C05454=1069.423,168.035,-78.116,173.237,27.810,155.027
C05455=1069.428,168.284,-78.138,173.240,27.813,155.027
C05456=1069.434,168.532,-78.160,173.242,27.815,155.028
C05457=1069.440,168.782,-78.182,173.243,27.818,155.028
C05458=1069.445,169.031,-78.205,173.246,27.821,155.028
C05459=1069.452,169.280,-78.227,173.247,27.824,155.029
C05460=1069.457,169.528,-78.250,173.250,27.827,155.029
C05461=1069.462,169.778,-78.272,173.251,27.830,155.030
C05462=1069.468,170.027,-78.294,173.253,27.832,155.030
C05463=1069.473,170.275,-78.316,173.255,27.835,155.030
C05464=1069.479,170.525,-78.338,173.257,27.838,155.031
C05465=1069.485,170.773,-78.361,173.259,27.841,155.031
C05466=1069.491,171.023,-78.383,173.261,27.844,155.032
C05467=1069.496,171.271,-78.405,173.263,27.847,155.032
C05468=1069.502,171.520,-78.427,173.265,27.850,155.032
C05469=1069.508,171.769,-78.450,173.266,27.852,155.033
C05470=1069.513,172.019,-78.472,173.269,27.855,155.033
C05471=1069.519,172.267,-78.495,173.270,27.858,155.034
C05472=1069.525,172.515,-78.517,173.273,27.861,155.034
C05473=1069.530,172.765,-78.539,173.274,27.864,155.034
C05474=1069.536,173.014,-78.562,173.277,27.867,155.035
C05475=1069.542,173.263,-78.584,173.278,27.870,155.035
C05476=1069.548,173.512,-78.607,173.280,27.872,155.036
C05477=1069.553,173.760,-78.630,173.282,27.875,155.036
C05478=1069.558,174.010,-78.652,173.284,27.878,155.036
C05479=1069.565,174.258,-78.674,173.286,27.881,155.037
C05480=1069.570,174.508,-78.696,173.288,27.884,155.037
C05481=1069.576,174.790,-78.722,173.290,27.887,155.037
C05482=1069.583,175.072,-78.747,173.293,27.890,155.038
C05483=1069.590,175.355,-78.774,173.295,27.893,155.038
C05484=1069.597,175.637,-78.799,173.297,27.897,155.039
C05485=1069.602,175.886,-78.821,173.299,27.900,155.039
C05486=1069.608,176.135,-78.844,173.301,27.902,155.040
C05487=1069.614,176.383,-78.866,173.303,27.905,155.040
C05488=1069.619,176.633,-78.888,173.305,27.908,155.040
C05489=1069.625,176.881,-78.911,173.307,27.911,155.041
C05490=1069.631,177.130,-78.934,173.309,27.913,155.041
C05491=1069.637,177.379,-78.957,173.311,27.916,155.042
C05492=1069.642,177.628,-78.979,173.313,27.919,155.042
C05493=1069.648,177.877,-79.002,173.315,27.922,155.042
C05494=1069.654,178.126,-79.025,173.317,27.925,155.043
C05495=1069.660,178.375,-79.048,173.319,27.928,155.043
C05496=1069.666,178.624,-79.070,173.321,27.931,155.044
C05497=1069.672,178.873,-79.092,173.323,27.933,155.044
C05498=1069.677,179.122,-79.115,173.325,27.936,155.044
C05499=1069.682,179.370,-79.138,173.327,27.939,155.045
C05500=1069.688,179.619,-79.161,173.329,27.942,155.045
C05501=1069.695,179.868,-79.183,173.331,27.945,155.046
C05502=1069.700,180.117,-79.206,173.333,27.948,155.046
C05503=1069.706,180.366,-79.229,173.335,27.950,155.046
C05504=1069.711,180.615,-79.251,173.337,27.953,155.047
C05505=1069.717,180.864,-79.274,173.339,27.956,155.047
C05506=1069.724,181.113,-79.296,173.341,27.959,155.048
C05507=1069.729,181.361,-79.319,173.343,27.961,155.048
C05508=1069.735,181.610,-79.342,173.345,27.964,155.048
C05509=1069.741,181.859,-79.365,173.348,27.967,155.049
C05510=1069.747,182.108,-79.388,173.349,27.970,155.049
C05511=1069.753,182.357,-79.411,173.352,27.973,155.049
C05512=1069.759,182.606,-79.434,173.353,27.976,155.050
C05513=1069.765,182.855,-79.456,173.356,27.979,155.050
C05514=1069.770,183.103,-79.479,173.357,27.982,155.051
C05515=1069.777,183.353,-79.503,173.360,27.985,155.051
C05516=1069.782,183.602,-79.526,173.362,27.987,155.051
C05517=1069.788,183.851,-79.549,173.364,27.990,155.052
C05518=1069.795,184.099,-79.571,173.366,27.993,155.052
C05519=1069.800,184.348,-79.594,173.368,27.995,155.052
C05520=1069.806,184.597,-79.617,173.370,27.998,155.053
C05521=1069.812,184.846,-79.640,173.372,28.001,155.053
C05522=1069.817,185.095,-79.663,173.374,28.004,155.054
C05523=1069.822,185.344,-79.686,173.376,28.007,155.054
C05524=1069.828,185.593,-79.709,173.378,28.010,155.055
C05525=1069.834,185.841,-79.733,173.380,28.013,155.055
C05526=1069.839,186.091,-79.756,173.382,28.016,155.055
C05527=1069.845,186.339,-79.779,173.384,28.019,155.056
C05528=1069.851,186.588,-79.802,173.387,28.022,155.056
C05529=1069.856,186.837,-79.825,173.388,28.025,155.057
C05530=1069.861,187.087,-79.849,173.391,28.028,155.057
C05531=1069.867,187.335,-79.872,173.392,28.031,155.057
C05532=1069.873,187.584,-79.895,173.395,28.034,155.058
C05533=1069.878,187.833,-79.919,173.396,28.037,155.058
C05534=1069.884,188.082,-79.942,173.399,28.040,155.059
C05535=1069.890,188.331,-79.965,173.400,28.043,155.059
C05536=1069.896,188.579,-79.989,173.403,28.046,155.060
C05537=1069.901,188.828,-80.012,173.404,28.049,155.060
C05538=1069.906,189.077,-80.035,173.407,28.052,155.060
C05539=1069.912,189.325,-80.059,173.409,28.055,155.061
C05540=1069.917,189.575,-80.082,173.411,28.058,155.061
C05541=1069.923,189.823,-80.105,173.413,28.061,155.062
C05542=1069.929,190.072,-80.128,173.415,28.063,155.062
C05543=1069.934,190.321,-80.152,173.417,28.067,155.063
C05544=1069.940,190.570,-80.175,173.419,28.070,155.063
C05545=1069.946,190.852,-80.202,173.421,28.073,155.063
C05546=1069.952,191.133,-80.228,173.424,28.076,155.064
C05547=1069.959,191.416,-80.255,173.426,28.080,155.064
C05548=1069.965,191.698,-80.282,173.429,28.083,155.065
C05549=1069.971,191.946,-80.305,173.431,28.086,155.065
C05550=1069.977,192.195,-80.328,173.433,28.089,155.066
C05551=1069.982,192.444,-80.352,173.435,28.092,155.066
C05552=1069.988,192.693,-80.376,173.438,28.095,155.066
C05553=1069.994,192.942,-80.399,173.439,28.098,155.067
C05554=1069.999,193.191,-80.423,173.442,28.101,155.067
C05555=1070.005,193.440,-80.446,173.443,28.104,155.068
C05556=1070.011,193.688,-80.470,173.446,28.107,155.068
C05557=1070.016,193.937,-80.493,173.448,28.110,155.069
C05558=1070.022,194.185,-80.517,173.450,28.113,155.069
C05559=1070.027,194.435,-80.540,173.452,28.116,155.069
C05560=1070.034,194.684,-80.565,173.454,28.119,155.070
C05561=1070.040,194.933,-80.587,173.456,28.122,155.070
C05562=1070.045,195.181,-80.612,173.459,28.125,155.071
C05563=1070.051,195.430,-80.635,173.460,28.128,155.071
C05564=1070.056,195.679,-80.659,173.463,28.131,155.072
C05565=1070.062,195.928,-80.682,173.464,28.134,155.072
C05566=1070.068,196.176,-80.706,173.467,28.137,155.072
C05567=1070.074,196.425,-80.730,173.469,28.140,155.073
C05568=1070.079,196.674,-80.753,173.471,28.142,155.073
C05569=1070.085,196.923,-80.777,173.474,28.145,155.074
C05570=1070.091,197.172,-80.801,173.476,28.149,155.074
C05571=1070.097,197.420,-80.824,173.478,28.152,155.074
C05572=1070.102,197.669,-80.849,173.480,28.155,155.075
C05573=1070.108,197.918,-80.872,173.483,28.158,155.075
C05574=1070.114,198.167,-80.896,173.484,28.160,155.076
C05575=1070.120,198.415,-80.920,173.487,28.163,155.076
C05576=1070.125,198.665,-80.943,173.488,28.167,155.077
C05577=1070.131,198.913,-80.967,173.491,28.170,155.077
C05578=1070.137,199.162,-80.992,173.493,28.173,155.077
C05579=1070.143,199.411,-81.015,173.495,28.175,155.078
C05580=1070.149,199.659,-81.038,173.497,28.178,155.078
C05581=1070.154,199.909,-81.063,173.500,28.181,155.079
C05582=1070.161,200.157,-81.087,173.501,28.184,155.079
C05583=1070.166,200.406,-81.111,173.504,28.187,155.079
C05584=1070.172,200.655,-81.134,173.506,28.190,155.080
C05585=1070.177,200.904,-81.158,173.508,28.193,155.080
C05586=1070.183,201.152,-81.182,173.510,28.196,155.081
C05587=1070.189,201.401,-81.207,173.513,28.200,155.081
C05588=1070.195,201.650,-81.230,173.515,28.203,155.082
C05589=1070.200,201.899,-81.254,173.517,28.205,155.082
C05590=1070.207,202.148,-81.278,173.519,28.208,155.082
C05591=1070.212,202.396,-81.302,173.522,28.211,155.083
C05592=1070.218,202.645,-81.326,173.523,28.214,155.083
C05593=1070.224,202.894,-81.350,173.526,28.217,155.084
C05594=1070.230,203.143,-81.375,173.528,28.220,155.084
C05595=1070.235,203.391,-81.399,173.530,28.224,155.085
C05596=1070.241,203.639,-81.423,173.533,28.227,155.085
C05597=1070.247,203.889,-81.446,173.535,28.230,155.085
C05598=1070.252,204.138,-81.471,173.537,28.233,155.086
C05599=1070.257,204.386,-81.495,173.539,28.236,155.086
C05600=1070.264,204.635,-81.519,173.542,28.239,155.087
C05601=1070.269,204.884,-81.543,173.543,28.242,155.087
C05602=1070.274,205.133,-81.568,173.546,28.245,155.088
C05603=1070.280,205.382,-81.592,173.548,28.248,155.088
C05604=1070.286,205.630,-81.616,173.551,28.251,155.088
C05605=1070.292,205.879,-81.640,173.552,28.254,155.089
C05606=1070.297,206.128,-81.665,173.555,28.258,155.089
C05607=1070.303,206.377,-81.689,173.557,28.261,155.090
C05608=1070.309,206.625,-81.714,173.559,28.263,155.090
C05609=1070.338,207.881,-81.837,173.698,28.338,155.093
C05610=1070.343,208.093,-81.858,173.701,28.341,155.094
C05611=1070.348,208.306,-81.880,173.702,28.344,155.094
C05612=1070.353,208.518,-81.901,173.704,28.348,155.095
C05613=1070.359,208.731,-81.923,173.705,28.352,155.096
C05614=1070.363,208.944,-81.944,173.707,28.355,155.096
C05615=1070.368,209.156,-81.966,173.709,28.358,155.097
C05616=1070.373,209.369,-81.987,173.710,28.361,155.097
C05617=1070.379,209.618,-82.012,173.713,28.366,155.098
C05618=1070.385,209.866,-82.037,173.714,28.369,155.099
C05619=1070.391,210.115,-82.062,173.717,28.373,155.099
C05620=1070.397,210.364,-82.087,173.719,28.378,155.100
C05621=1070.402,210.612,-82.113,173.720,28.382,155.101
C05622=1070.409,210.861,-82.138,173.723,28.386,155.101
C05623=1070.414,211.110,-82.163,173.725,28.390,155.102
C05624=1070.420,211.358,-82.188,173.726,28.394,155.103
C05625=1070.426,211.607,-82.213,173.729,28.398,155.103
C05626=1070.432,211.856,-82.239,173.731,28.402,155.104
C05627=1070.437,212.104,-82.264,173.733,28.405,155.104
C05628=1070.444,212.353,-82.289,173.735,28.410,155.105
C05629=1070.449,212.602,-82.314,173.737,28.414,155.106
C05630=1070.456,212.851,-82.339,173.739,28.417,155.106
C05631=1070.461,213.099,-82.365,173.741,28.421,155.107
C05632=1070.467,213.348,-82.390,173.744,28.425,155.108
C05633=1070.473,213.596,-82.416,173.745,28.430,155.108
C05634=1070.478,213.845,-82.442,173.747,28.434,155.109
C05635=1070.484,214.093,-82.467,173.750,28.438,155.110
C05636=1070.490,214.342,-82.492,173.751,28.442,155.110
C05637=1070.496,214.591,-82.518,173.754,28.446,155.111
C05638=1070.502,214.840,-82.543,173.756,28.450,155.112
C05639=1070.508,215.088,-82.568,173.757,28.453,155.112
C05640=1070.513,215.336,-82.594,173.760,28.457,155.113
C05641=1070.519,215.585,-82.619,173.762,28.462,155.114
C05642=1070.525,215.834,-82.645,173.764,28.465,155.114
C05643=1070.531,216.083,-82.671,173.766,28.469,155.115
C05644=1070.537,216.331,-82.696,173.768,28.474,155.116
C05645=1070.543,216.580,-82.722,173.770,28.478,155.116
C05646=1070.548,216.828,-82.747,173.772,28.482,155.117
C05647=1070.554,217.077,-82.772,173.775,28.486,155.118
C05648=1070.560,217.326,-82.798,173.776,28.490,155.118
C05649=1070.566,217.575,-82.824,173.778,28.494,155.119
C05650=1070.572,217.823,-82.850,173.781,28.498,155.119
C05651=1070.578,218.072,-82.875,173.783,28.502,155.120
C05652=1070.584,218.320,-82.901,173.785,28.505,155.121
C05653=1070.590,218.569,-82.927,173.787,28.509,155.121
C05654=1070.595,218.817,-82.952,173.789,28.513,155.122
C05655=1070.601,219.066,-82.978,173.791,28.517,155.123
C05656=1070.607,219.314,-83.004,173.793,28.521,155.123
C05657=1070.613,219.563,-83.029,173.796,28.525,155.124
C05658=1070.619,219.812,-83.055,173.798,28.529,155.125
C05659=1070.625,220.061,-83.080,173.799,28.533,155.125
C05660=1070.631,220.310,-83.106,173.802,28.537,155.126
C05661=1070.637,220.558,-83.132,173.804,28.541,155.127
C05662=1070.643,220.807,-83.158,173.806,28.545,155.127
C05663=1070.649,221.055,-83.184,173.808,28.549,155.128
C05664=1070.655,221.304,-83.209,173.811,28.553,155.129
C05665=1070.660,221.519,-83.232,173.812,28.556,155.129
C05666=1070.665,221.733,-83.254,173.815,28.560,155.130
C05667=1070.670,221.948,-83.277,173.816,28.563,155.130
C05668=1070.675,222.163,-83.298,173.817,28.567,155.131
C05669=1070.680,222.379,-83.322,173.820,28.570,155.131
C05670=1070.685,222.593,-83.344,173.821,28.573,155.132
C05671=1070.690,222.808,-83.367,173.823,28.577,155.132
C05672=1070.695,223.022,-83.389,173.825,28.580,155.133
C05673=1070.701,223.271,-83.415,173.827,28.584,155.134
C05674=1070.707,223.520,-83.440,173.829,28.588,155.134
C05675=1070.713,223.768,-83.467,173.832,28.592,155.135
C05676=1070.718,224.017,-83.493,173.834,28.596,155.136
C05677=1070.725,224.265,-83.519,173.836,28.600,155.136
C05678=1070.730,224.514,-83.545,173.838,28.604,155.137
C05679=1070.736,224.763,-83.571,173.840,28.608,155.138
C05680=1070.741,225.012,-83.597,173.843,28.612,155.138
C05681=1070.748,225.260,-83.623,173.844,28.616,155.139
C05682=1070.753,225.509,-83.649,173.847,28.620,155.139
C05683=1070.759,225.757,-83.676,173.849,28.624,155.140
C05684=1070.765,226.006,-83.701,173.851,28.628,155.141
C05685=1070.771,226.254,-83.728,173.853,28.632,155.141
C05686=1070.776,226.503,-83.754,173.855,28.636,155.142
C05687=1070.783,226.751,-83.780,173.858,28.640,155.143
C05688=1070.788,227.000,-83.806,173.860,28.644,155.143
C05689=1070.794,227.248,-83.833,173.862,28.648,155.144
C05690=1070.800,227.497,-83.859,173.864,28.652,155.145
C05691=1070.806,227.745,-83.885,173.866,28.656,155.145
C05692=1070.812,227.994,-83.911,173.869,28.659,155.146
C05693=1070.817,228.243,-83.937,173.870,28.663,155.146
C05694=1070.825,228.492,-83.964,173.873,28.667,155.147
C05695=1070.830,228.740,-83.990,173.875,28.671,155.148
C05696=1070.836,228.989,-84.016,173.878,28.675,155.148
C05697=1070.842,229.237,-84.043,173.880,28.679,155.149
C05698=1070.848,229.485,-84.069,173.882,28.683,155.150
C05699=1070.854,229.734,-84.095,173.884,28.687,155.150
C05700=1070.859,229.983,-84.121,173.886,28.691,155.151
C05701=1070.865,230.231,-84.148,173.889,28.695,155.152
C05702=1070.871,230.480,-84.175,173.891,28.699,155.152
C05703=1070.877,230.729,-84.201,173.893,28.702,155.153
C05704=1070.883,230.977,-84.228,173.895,28.706,155.154
C05705=1070.888,231.226,-84.254,173.898,28.710,155.154
C05706=1070.894,231.474,-84.281,173.900,28.714,155.155
C05707=1070.901,231.722,-84.307,173.901,28.718,155.155
C05708=1070.906,231.971,-84.333,173.904,28.722,155.156
C05709=1070.912,232.220,-84.360,173.906,28.726,155.157
C05710=1070.918,232.469,-84.387,173.909,28.730,155.157
C05711=1070.924,232.717,-84.413,173.911,28.734,155.158
C05712=1070.930,232.965,-84.440,173.913,28.738,155.159
C05713=1070.936,233.214,-84.467,173.915,28.742,155.159
C05714=1070.941,233.462,-84.493,173.917,28.746,155.160
C05715=1070.947,233.710,-84.520,173.920,28.750,155.161
C05716=1070.953,233.960,-84.546,173.922,28.754,155.161
C05717=1070.959,234.208,-84.573,173.925,28.758,155.162
C05718=1070.965,234.457,-84.599,173.926,28.762,155.163
C05719=1070.971,234.705,-84.626,173.929,28.766,155.163
C05720=1070.976,234.954,-84.653,173.931,28.770,155.164
C05721=1070.981,235.165,-84.676,173.933,28.773,155.164
C05722=1070.986,235.375,-84.698,173.935,28.776,155.165
C05723=1070.991,235.586,-84.722,173.937,28.779,155.165
C05724=1070.996,235.797,-84.744,173.939,28.783,155.166
C05725=1071.001,236.008,-84.767,173.941,28.787,155.167
C05726=1071.006,236.219,-84.789,173.942,28.790,155.167
C05727=1071.011,236.429,-84.812,173.945,28.793,155.168
C05728=1071.016,236.640,-84.836,173.946,28.796,155.168
C05729=1071.022,236.888,-84.862,173.949,28.800,155.169
C05730=1071.028,237.136,-84.889,173.951,28.804,155.170
C05731=1071.033,237.385,-84.916,173.954,28.808,155.170
C05732=1071.040,237.634,-84.943,173.955,28.812,155.171
C05733=1071.045,237.882,-84.969,173.957,28.816,155.172
C05734=1071.050,238.131,-84.997,173.960,28.820,155.172
C05735=1071.057,238.380,-85.024,173.962,28.824,155.173
C05736=1071.063,238.628,-85.051,173.965,28.828,155.173
C05737=1071.069,238.876,-85.078,173.967,28.832,155.174
C05738=1071.074,239.124,-85.104,173.970,28.835,155.175
C05739=1071.081,239.374,-85.131,173.971,28.839,155.175
C05740=1071.087,239.622,-85.158,173.974,28.843,155.176
C05741=1071.092,239.870,-85.186,173.976,28.847,155.177
C05742=1071.098,240.119,-85.213,173.979,28.851,155.177
C05743=1071.104,240.367,-85.240,173.981,28.855,155.178
C05744=1071.110,240.616,-85.266,173.983,28.859,155.178
C05745=1071.117,240.864,-85.294,173.986,28.863,155.179
C05746=1071.122,241.113,-85.321,173.987,28.867,155.180
C05747=1071.127,241.361,-85.348,173.990,28.871,155.180
C05748=1071.134,241.610,-85.376,173.992,28.875,155.181
C05749=1071.140,241.858,-85.402,173.995,28.879,155.182
C05750=1071.146,242.106,-85.429,173.997,28.883,155.182
C05751=1071.152,242.355,-85.457,174.000,28.887,155.183
C05752=1071.157,242.603,-85.484,174.002,28.890,155.184
C05753=1071.163,242.851,-85.511,174.005,28.894,155.184
C05754=1071.169,243.101,-85.539,174.006,28.898,155.185
C05755=1071.175,243.349,-85.565,174.009,28.902,155.185
C05756=1071.180,243.597,-85.593,174.011,28.906,155.186
C05757=1071.187,243.846,-85.620,174.013,28.910,155.187
C05758=1071.193,244.094,-85.648,174.016,28.914,155.188
C05759=1071.198,244.342,-85.675,174.018,28.918,155.188
C05760=1071.204,244.591,-85.703,174.021,28.922,155.189
C05761=1071.209,244.840,-85.730,174.023,28.926,155.189
C05762=1071.216,245.088,-85.758,174.026,28.930,155.190
C05763=1071.221,245.337,-85.785,174.027,28.934,155.191
C05764=1071.227,245.584,-85.812,174.030,28.938,155.191
C05765=1071.234,245.833,-85.839,174.032,28.941,155.192
C05766=1071.239,246.082,-85.867,174.035,28.945,155.193
C05767=1071.246,246.330,-85.895,174.037,28.949,155.193
C05768=1071.251,246.579,-85.922,174.039,28.953,155.194
C05769=1071.257,246.827,-85.950,174.042,28.957,155.194
C05770=1071.262,247.076,-85.977,174.044,28.961,155.195
C05771=1071.268,247.324,-86.005,174.047,28.966,155.196
C05772=1071.274,247.572,-86.033,174.049,28.970,155.197
C05773=1071.279,247.821,-86.060,174.051,28.973,155.197
C05774=1071.285,248.069,-86.088,174.053,28.977,155.198
C05775=1071.291,248.317,-86.116,174.056,28.981,155.199
C05776=1071.297,248.565,-86.144,174.058,28.985,155.199
C05777=1071.306,248.981,-86.189,174.062,28.992,155.200
C05778=1071.316,249.396,-86.237,174.066,28.999,155.201
C05779=1071.326,249.811,-86.283,174.070,29.005,155.202
C05780=1071.335,250.226,-86.329,174.074,29.012,155.204
C05781=1071.341,250.474,-86.357,174.077,29.016,155.204
C05782=1071.347,250.723,-86.385,174.079,29.020,155.205
C05783=1071.353,250.971,-86.412,174.082,29.024,155.206
C05784=1071.359,251.220,-86.441,174.084,29.028,155.206
C05785=1071.365,251.467,-86.468,174.086,29.032,155.207
C05786=1071.371,251.716,-86.496,174.088,29.036,155.207
C05787=1071.376,251.965,-86.524,174.091,29.040,155.208
C05788=1071.382,252.213,-86.551,174.093,29.044,155.209
C05789=1071.388,252.461,-86.579,174.096,29.048,155.209
C05790=1071.394,252.710,-86.608,174.098,29.052,155.210
C05791=1071.399,252.958,-86.636,174.101,29.056,155.211
C05792=1071.406,253.207,-86.663,174.103,29.060,155.211
C05793=1071.412,253.455,-86.692,174.106,29.064,155.212
C05794=1071.417,253.703,-86.720,174.108,29.067,155.213
C05795=1071.423,253.952,-86.748,174.111,29.071,155.213
C05796=1071.429,254.200,-86.775,174.113,29.075,155.214
C05797=1071.435,254.449,-86.804,174.115,29.079,155.215
C05798=1071.440,254.697,-86.832,174.118,29.083,155.215
C05799=1071.446,254.945,-86.860,174.120,29.087,155.216
C05800=1071.453,255.194,-86.888,174.123,29.091,155.217
C05801=1071.458,255.442,-86.916,174.125,29.095,155.217
C05802=1071.464,255.691,-86.944,174.128,29.099,155.218
C05803=1071.470,255.938,-86.973,174.130,29.103,155.218
C05804=1071.476,256.186,-87.000,174.133,29.107,155.219
C05805=1071.482,256.435,-87.029,174.135,29.111,155.220
C05806=1071.488,256.683,-87.057,174.138,29.115,155.220
C05807=1071.494,256.932,-87.085,174.140,29.119,155.221
C05808=1071.500,257.181,-87.113,174.143,29.123,155.222
C05809=1071.506,257.429,-87.141,174.145,29.127,155.222
C05810=1071.512,257.677,-87.170,174.148,29.131,155.223
C05811=1071.518,257.925,-87.198,174.150,29.135,155.224
C05812=1071.523,258.173,-87.226,174.153,29.138,155.224
C05813=1071.529,258.422,-87.254,174.155,29.142,155.225
C05814=1071.535,258.670,-87.283,174.158,29.146,155.225
C05815=1071.541,258.918,-87.311,174.160,29.150,155.226
C05816=1071.547,259.167,-87.339,174.163,29.154,155.227
C05817=1071.553,259.416,-87.367,174.165,29.158,155.227
C05818=1071.560,259.664,-87.396,174.168,29.162,155.228
C05819=1071.565,259.912,-87.424,174.170,29.166,155.229
C05820=1071.571,260.161,-87.453,174.173,29.170,155.229
C05821=1071.578,260.408,-87.481,174.175,29.173,155.230
C05822=1071.584,260.657,-87.510,174.178,29.177,155.231
C05823=1071.589,260.905,-87.537,174.180,29.181,155.231
C05824=1071.595,261.153,-87.567,174.183,29.185,155.232
C05825=1071.601,261.402,-87.595,174.185,29.189,155.233
C05826=1071.608,261.650,-87.624,174.187,29.193,155.233
C05827=1071.614,261.899,-87.652,174.190,29.197,155.234
C05828=1071.620,262.147,-87.680,174.193,29.200,155.234
C05829=1071.630,262.559,-87.727,174.197,29.207,155.235
C05830=1071.640,262.971,-87.775,174.201,29.214,155.237
C05831=1071.651,263.385,-87.822,174.205,29.220,155.238
C05832=1071.661,263.797,-87.870,174.209,29.227,155.239
C05833=1071.665,264.045,-87.899,174.212,29.231,155.239
C05834=1071.671,264.294,-87.927,174.214,29.235,155.240
C05835=1071.678,264.542,-87.956,174.217,29.239,155.241
C05836=1071.684,264.791,-87.985,174.219,29.242,155.241
C05837=1071.690,265.039,-88.014,174.223,29.247,155.242
C05838=1071.695,265.286,-88.043,174.225,29.251,155.243
C05839=1071.701,265.535,-88.071,174.228,29.254,155.243
C05840=1071.707,265.783,-88.100,174.230,29.258,155.244
C05841=1071.713,266.031,-88.129,174.233,29.262,155.245
C05842=1071.719,266.280,-88.158,174.235,29.266,155.245
C05843=1071.725,266.528,-88.186,174.238,29.270,155.246
C05844=1071.730,266.776,-88.216,174.240,29.274,155.246
C05845=1071.736,267.025,-88.244,174.243,29.278,155.247
C05846=1071.743,267.273,-88.273,174.245,29.282,155.248
C05847=1071.749,267.521,-88.302,174.248,29.286,155.249
C05848=1071.754,267.769,-88.332,174.250,29.290,155.249
C05849=1071.760,268.018,-88.360,174.253,29.294,155.250
C05850=1071.766,268.266,-88.389,174.255,29.298,155.251
C05851=1071.772,268.514,-88.418,174.258,29.302,155.251
C05852=1071.778,268.762,-88.447,174.261,29.306,155.252
C05853=1071.784,269.010,-88.477,174.264,29.310,155.252
C05854=1071.790,269.258,-88.506,174.266,29.314,155.253
C05855=1071.796,269.507,-88.534,174.269,29.318,155.254
C05856=1071.802,269.756,-88.564,174.271,29.322,155.254
C05857=1071.808,270.004,-88.593,174.274,29.326,155.255
C05858=1071.814,270.252,-88.622,174.276,29.330,155.256
C05859=1071.819,270.500,-88.651,174.279,29.334,155.256
C05860=1071.825,270.748,-88.680,174.281,29.338,155.257
C05861=1071.831,270.996,-88.709,174.284,29.342,155.258
C05862=1071.837,271.244,-88.739,174.286,29.346,155.258
C05863=1071.843,271.493,-88.768,174.290,29.350,155.259
C05864=1071.849,271.741,-88.798,174.292,29.354,155.260
C05865=1071.855,271.989,-88.827,174.295,29.358,155.260
C05866=1071.861,272.237,-88.856,174.297,29.362,155.261
C05867=1071.867,272.486,-88.885,174.300,29.366,155.262
C05868=1071.873,272.734,-88.914,174.302,29.370,155.262
C05869=1071.879,272.982,-88.944,174.305,29.374,155.263
C05870=1071.885,273.230,-88.973,174.307,29.378,155.264
C05871=1071.891,273.479,-89.002,174.310,29.382,155.264
C05872=1071.897,273.727,-89.032,174.313,29.386,155.265
C05873=1071.903,273.974,-89.061,174.316,29.390,155.266
C05874=1071.909,274.223,-89.091,174.318,29.394,155.266
C05875=1071.915,274.471,-89.120,174.321,29.398,155.267
C05876=1071.920,274.719,-89.150,174.323,29.402,155.268
C05877=1071.926,274.968,-89.179,174.326,29.406,155.268
C05878=1071.932,275.216,-89.208,174.328,29.410,155.269
C05879=1071.938,275.464,-89.239,174.332,29.414,155.270
C05880=1071.944,275.712,-89.268,174.334,29.418,155.270
C05881=1071.953,276.128,-89.317,174.338,29.425,155.271
C05882=1071.964,276.544,-89.367,174.342,29.432,155.273
C05883=1071.973,276.959,-89.417,174.347,29.438,155.274
C05884=1071.983,277.375,-89.466,174.352,29.445,155.275
C05885=1071.989,277.623,-89.496,174.354,29.449,155.276
C05886=1071.995,277.871,-89.525,174.357,29.453,155.276
C05887=1072.001,278.120,-89.555,174.359,29.457,155.277
C05888=1072.007,278.368,-89.586,174.362,29.461,155.278
C05889=1072.014,278.616,-89.615,174.365,29.465,155.278
C05890=1072.019,278.864,-89.645,174.368,29.470,155.279
C05891=1072.025,279.113,-89.675,174.370,29.474,155.280
C05892=1072.031,279.361,-89.704,174.373,29.477,155.280
C05893=1072.037,279.609,-89.734,174.375,29.481,155.281
C05894=1072.043,279.857,-89.764,174.378,29.485,155.282
C05895=1072.049,280.105,-89.793,174.381,29.490,155.282
C05896=1072.055,280.353,-89.823,174.384,29.494,155.283
C05897=1072.061,280.602,-89.854,174.386,29.498,155.284
C05898=1072.067,280.850,-89.883,174.389,29.502,155.284
C05899=1072.073,281.098,-89.913,174.391,29.506,155.285
C05900=1072.079,281.345,-89.943,174.394,29.510,155.286
C05901=1072.084,281.594,-89.973,174.397,29.514,155.286
C05902=1072.090,281.842,-90.003,174.400,29.518,155.287
C05903=1072.096,282.090,-90.033,174.402,29.522,155.288
C05904=1072.102,282.338,-90.063,174.405,29.526,155.288
C05905=1072.109,282.586,-90.094,174.408,29.530,155.289
C05906=1072.114,282.835,-90.123,174.411,29.535,155.290
C05907=1072.120,283.082,-90.154,174.414,29.539,155.290
C05908=1072.126,283.330,-90.184,174.416,29.543,155.291
C05909=1072.131,283.579,-90.214,174.419,29.546,155.292
C05910=1072.137,283.826,-90.244,174.421,29.551,155.293
C05911=1072.144,284.075,-90.275,174.425,29.555,155.293
C05912=1072.149,284.323,-90.305,174.427,29.559,155.294
C05913=1072.155,284.571,-90.335,174.430,29.563,155.295
C05914=1072.162,284.819,-90.364,174.432,29.567,155.295
C05915=1072.167,285.067,-90.395,174.436,29.571,155.296
C05916=1072.174,285.315,-90.425,174.438,29.576,155.297
C05917=1072.180,285.563,-90.456,174.441,29.580,155.297
C05918=1072.185,285.811,-90.485,174.443,29.583,155.298
C05919=1072.191,286.059,-90.516,174.446,29.587,155.299
C05920=1072.197,286.308,-90.546,174.449,29.592,155.299
C05921=1072.203,286.555,-90.577,174.452,29.596,155.300
C05922=1072.209,286.803,-90.607,174.454,29.600,155.301
C05923=1072.215,287.051,-90.638,174.457,29.604,155.302
C05924=1072.221,287.300,-90.668,174.460,29.608,155.302
C05925=1072.227,287.547,-90.699,174.463,29.612,155.303
C05926=1072.233,287.795,-90.729,174.465,29.617,155.304
C05927=1072.239,288.044,-90.760,174.468,29.620,155.304
C05928=1072.246,288.291,-90.789,174.471,29.625,155.305
C05929=1072.252,288.539,-90.820,174.474,29.628,155.306
C05930=1072.257,288.787,-90.850,174.476,29.633,155.306
C05931=1072.264,289.035,-90.881,174.479,29.637,155.307
C05932=1072.269,289.284,-90.912,174.483,29.641,155.308
C05933=1072.274,289.497,-90.937,174.484,29.644,155.308
C05934=1072.279,289.710,-90.964,174.487,29.648,155.309
C05935=1072.285,289.923,-90.990,174.489,29.652,155.310
C05936=1072.289,290.136,-91.016,174.492,29.655,155.310
C05937=1072.295,290.349,-91.043,174.494,29.659,155.311
C05938=1072.300,290.562,-91.069,174.496,29.662,155.311
C05939=1072.305,290.774,-91.095,174.499,29.666,155.312
C05940=1072.310,290.989,-91.122,174.501,29.669,155.312
C05941=1072.316,291.236,-91.153,174.504,29.674,155.313
C05942=1072.322,291.484,-91.183,174.507,29.678,155.314
C05943=1072.328,291.732,-91.214,174.510,29.682,155.315
C05944=1072.334,291.980,-91.244,174.512,29.686,155.315
C05945=1072.340,292.228,-91.275,174.515,29.690,155.316
C05946=1072.346,292.476,-91.307,174.518,29.694,155.317
C05947=1072.352,292.724,-91.337,174.521,29.698,155.317
C05948=1072.358,292.972,-91.368,174.523,29.703,155.318
C05949=1072.364,293.219,-91.399,174.527,29.707,155.319
C05950=1072.369,293.468,-91.430,174.529,29.711,155.320
C05951=1072.376,293.716,-91.460,174.532,29.715,155.320
C05952=1072.381,293.964,-91.491,174.535,29.720,155.321
C05953=1072.388,294.212,-91.522,174.538,29.724,155.322
C05954=1072.394,294.460,-91.553,174.541,29.728,155.322
C05955=1072.400,294.708,-91.585,174.543,29.732,155.323
C05956=1072.406,294.956,-91.615,174.547,29.736,155.324
C05957=1072.412,295.204,-91.645,174.549,29.740,155.325
C05958=1072.418,295.452,-91.677,174.552,29.745,155.325
C05959=1072.423,295.700,-91.708,174.555,29.749,155.326
C05960=1072.430,295.947,-91.739,174.558,29.753,155.327
C05961=1072.435,296.196,-91.770,174.560,29.757,155.327
C05962=1072.442,296.444,-91.801,174.564,29.762,155.328
C05963=1072.448,296.691,-91.832,174.566,29.766,155.329
C05964=1072.454,296.940,-91.864,174.569,29.770,155.330
C05965=1072.460,297.187,-91.894,174.572,29.774,155.330
C05966=1072.466,297.435,-91.926,174.575,29.778,155.331
C05967=1072.471,297.683,-91.957,174.577,29.782,155.332
C05968=1072.477,297.932,-91.989,174.581,29.787,155.332
C05969=1072.484,298.179,-92.020,174.583,29.791,155.333
C05970=1072.489,298.427,-92.051,174.586,29.796,155.334
C05971=1072.495,298.675,-92.082,174.590,29.800,155.335
C05972=1072.501,298.922,-92.114,174.592,29.804,155.335
C05973=1072.506,299.171,-92.145,174.595,29.808,155.336
C05974=1072.513,299.418,-92.176,174.598,29.813,155.337
C05975=1072.519,299.667,-92.208,174.601,29.817,155.338
C05976=1072.524,299.915,-92.239,174.603,29.821,155.338
C05977=1072.530,300.163,-92.271,174.607,29.826,155.339
C05978=1072.536,300.410,-92.302,174.609,29.830,155.340
C05979=1072.542,300.658,-92.334,174.612,29.834,155.341
C05980=1072.548,300.906,-92.365,174.615,29.839,155.341
C05981=1072.553,301.154,-92.397,174.618,29.843,155.342
C05982=1072.560,301.402,-92.428,174.621,29.847,155.343
C05983=1072.566,301.650,-92.460,174.624,29.852,155.344
C05984=1072.571,301.897,-92.491,174.626,29.856,155.344
C05985=1072.578,302.145,-92.523,174.630,29.861,155.345
C05986=1072.583,302.393,-92.554,174.632,29.864,155.346
C05987=1072.589,302.641,-92.586,174.635,29.869,155.347
C05988=1072.595,302.890,-92.618,174.638,29.873,155.347
C05989=1072.600,303.109,-92.646,174.641,29.877,155.348
C05990=1072.606,303.330,-92.673,174.644,29.881,155.349
C05991=1072.611,303.550,-92.702,174.646,29.885,155.349
C05992=1072.616,303.771,-92.730,174.649,29.889,155.350
C05993=1072.621,303.991,-92.759,174.651,29.893,155.351
C05994=1072.627,304.211,-92.787,174.654,29.896,155.351
C05995=1072.632,304.431,-92.815,174.657,29.900,155.352
C05996=1072.637,304.651,-92.843,174.659,29.904,155.353
C05997=1072.643,304.900,-92.875,174.662,29.908,155.353
C05998=1072.650,305.148,-92.907,174.665,29.913,155.354
C05999=1072.655,305.395,-92.938,174.668,29.917,155.355
C06000=1072.661,305.643,-92.970,174.671,29.921,155.356
C06001=1072.667,305.892,-93.002,174.674,29.926,155.356
C06002=1072.673,306.139,-93.034,174.677,29.930,155.357
C06003=1072.679,306.387,-93.066,174.680,29.935,155.358
C06004=1072.685,306.635,-93.098,174.682,29.939,155.359
C06005=1072.691,306.882,-93.130,174.686,29.943,155.359
C06006=1072.698,307.130,-93.161,174.689,29.948,155.360
C06007=1072.704,307.378,-93.193,174.692,29.952,155.361
C06008=1072.710,307.626,-93.225,174.695,29.957,155.362
C06009=1072.715,307.874,-93.257,174.698,29.961,155.362
C06010=1072.722,308.121,-93.289,174.701,29.965,155.363
C06011=1072.728,308.369,-93.321,174.704,29.969,155.364
C06012=1072.734,308.618,-93.353,174.707,29.974,155.365
C06013=1072.740,308.866,-93.385,174.709,29.978,155.366
C06014=1072.746,309.113,-93.418,174.713,29.983,155.366
C06015=1072.753,309.361,-93.449,174.715,29.987,155.367
C06016=1072.759,309.609,-93.481,174.719,29.991,155.368
C06017=1072.765,309.856,-93.514,174.721,29.996,155.369
C06018=1072.771,310.105,-93.546,174.725,30.000,155.369
C06019=1072.776,310.352,-93.578,174.728,30.004,155.370
C06020=1072.783,310.599,-93.610,174.731,30.009,155.371
C06021=1072.789,310.848,-93.642,174.734,30.013,155.371
C06022=1072.796,311.095,-93.675,174.737,30.017,155.372
C06023=1072.802,311.343,-93.707,174.740,30.022,155.373
C06024=1072.808,311.592,-93.739,174.743,30.026,155.374
C06025=1072.814,311.839,-93.771,174.746,30.031,155.375
C06026=1072.820,312.087,-93.803,174.749,30.035,155.375
C06027=1072.827,312.335,-93.836,174.752,30.040,155.376
C06028=1072.832,312.582,-93.867,174.755,30.044,155.377
C06029=1072.838,312.830,-93.900,174.758,30.048,155.378
C06030=1072.844,313.078,-93.932,174.762,30.053,155.378
C06031=1072.851,313.326,-93.965,174.764,30.057,155.379
C06032=1072.857,313.573,-93.997,174.768,30.061,155.380
C06033=1072.863,313.821,-94.029,174.770,30.066,155.381
C06034=1072.869,314.069,-94.062,174.774,30.070,155.381
C06035=1072.875,314.317,-94.094,174.776,30.075,155.382
C06036=1072.882,314.565,-94.127,174.780,30.079,155.383
C06037=1072.888,314.812,-94.160,174.782,30.084,155.384
C06038=1072.894,315.061,-94.192,174.786,30.088,155.385
C06039=1072.899,315.309,-94.225,174.788,30.093,155.386
C06040=1072.906,315.556,-94.258,174.792,30.098,155.386
C06041=1072.912,315.804,-94.291,174.795,30.102,155.387
C06042=1072.917,316.052,-94.323,174.798,30.106,155.388
C06043=1072.923,316.299,-94.356,174.801,30.111,155.389
C06044=1072.929,316.547,-94.388,174.804,30.116,155.390
C06045=1072.934,316.769,-94.418,174.807,30.120,155.390
C06046=1072.940,316.991,-94.448,174.809,30.124,155.391
C06047=1072.945,317.213,-94.476,174.812,30.128,155.392
C06048=1072.950,317.435,-94.506,174.815,30.132,155.392
C06049=1072.955,317.657,-94.536,174.817,30.137,155.393
C06050=1072.961,317.879,-94.565,174.820,30.140,155.394
C06051=1072.966,318.101,-94.594,174.823,30.145,155.395
C06052=1072.972,318.324,-94.624,174.826,30.149,155.395
C06053=1072.978,318.571,-94.657,174.828,30.154,155.396
C06054=1072.984,318.819,-94.691,174.832,30.158,155.397
C06055=1072.990,319.067,-94.723,174.835,30.162,155.398
C06056=1072.996,319.314,-94.756,174.838,30.168,155.399
C06057=1073.002,319.562,-94.789,174.841,30.172,155.400
C06058=1073.008,319.810,-94.822,174.844,30.176,155.400
C06059=1073.014,320.058,-94.855,174.848,30.181,155.401
C06060=1073.020,320.305,-94.888,174.850,30.186,155.402
C06061=1073.026,320.553,-94.921,174.854,30.190,155.403
C06062=1073.032,320.801,-94.954,174.856,30.195,155.404
C06063=1073.038,321.049,-94.987,174.860,30.200,155.404
C06064=1073.044,321.296,-95.020,174.862,30.204,155.405
C06065=1073.050,321.544,-95.053,174.866,30.209,155.406
C06066=1073.056,321.792,-95.086,174.869,30.213,155.407
C06067=1073.062,322.040,-95.119,174.872,30.219,155.408
C06068=1073.069,322.287,-95.153,174.876,30.223,155.409
C06069=1073.075,322.535,-95.186,174.878,30.227,155.409
C06070=1073.081,322.783,-95.219,174.882,30.232,155.410
C06071=1073.087,323.031,-95.252,174.884,30.237,155.411
C06072=1073.093,323.278,-95.285,174.888,30.242,155.412
C06073=1073.099,323.526,-95.319,174.891,30.246,155.413
C06074=1073.105,323.773,-95.352,174.894,30.251,155.414
C06075=1073.111,324.022,-95.386,174.897,30.256,155.414
C06076=1073.117,324.269,-95.418,174.900,30.261,155.415
C06077=1073.123,324.517,-95.452,174.904,30.265,155.416
C06078=1073.130,324.764,-95.485,174.907,30.270,155.417
C06079=1073.135,325.012,-95.519,174.910,30.274,155.418
C06080=1073.142,325.260,-95.552,174.913,30.279,155.419
C06081=1073.148,325.508,-95.586,174.916,30.284,155.419
C06082=1073.155,325.755,-95.619,174.919,30.288,155.420
C06083=1073.160,326.003,-95.652,174.923,30.293,155.421
C06084=1073.167,326.251,-95.686,174.925,30.298,155.422
C06085=1073.173,326.498,-95.720,174.929,30.303,155.423
C06086=1073.178,326.746,-95.753,174.933,30.307,155.424
C06087=1073.186,326.994,-95.787,174.935,30.312,155.425
C06088=1073.191,327.242,-95.820,174.939,30.317,155.425
C06089=1073.198,327.489,-95.854,174.942,30.322,155.426
C06090=1073.204,327.737,-95.887,174.945,30.326,155.427
C06091=1073.210,327.984,-95.921,174.948,30.331,155.428
C06092=1073.216,328.232,-95.954,174.951,30.336,155.429
C06093=1073.223,328.480,-95.988,174.955,30.340,155.430
C06094=1073.229,328.727,-96.022,174.958,30.345,155.431
C06095=1073.235,328.975,-96.055,174.961,30.350,155.431
C06096=1073.242,329.223,-96.089,174.964,30.355,155.432
C06097=1073.247,329.471,-96.122,174.968,30.360,155.433
C06098=1073.255,329.718,-96.156,174.970,30.364,155.434
C06099=1073.260,329.965,-96.190,174.974,30.369,155.435
C06100=1073.266,330.213,-96.224,174.977,30.374,155.436
C06101=1073.272,330.432,-96.253,174.980,30.378,155.436
C06102=1073.278,330.651,-96.284,174.983,30.382,155.437
C06103=1073.284,330.870,-96.314,174.986,30.387,155.438
C06104=1073.289,331.089,-96.343,174.989,30.391,155.439
C06105=1073.295,331.308,-96.373,174.992,30.395,155.439
C06106=1073.300,331.527,-96.403,174.994,30.399,155.440
C06107=1073.306,331.745,-96.433,174.998,30.404,155.441
C06108=1073.311,331.964,-96.464,175.000,30.408,155.442
C06109=1073.317,332.212,-96.497,175.004,30.413,155.443
C06110=1073.323,332.460,-96.531,175.006,30.418,155.444
C06111=1073.329,332.707,-96.565,175.010,30.423,155.445
C06112=1073.336,332.955,-96.600,175.014,30.428,155.445
C06113=1073.341,333.202,-96.634,175.016,30.433,155.446
C06114=1073.347,333.450,-96.668,175.020,30.438,155.447
C06115=1073.354,333.698,-96.702,175.023,30.443,155.448
C06116=1073.360,333.945,-96.736,175.027,30.448,155.449
C06117=1073.366,334.193,-96.771,175.029,30.452,155.450
C06118=1073.372,334.440,-96.805,175.033,30.457,155.451
C06119=1073.378,334.688,-96.839,175.036,30.463,155.452
C06120=1073.384,334.936,-96.873,175.039,30.467,155.453
C06121=1073.391,335.184,-96.908,175.043,30.472,155.454
C06122=1073.397,335.431,-96.942,175.046,30.477,155.454
C06123=1073.403,335.679,-96.976,175.050,30.482,155.455
C06124=1073.409,335.926,-97.010,175.052,30.487,155.456
C06125=1073.416,336.173,-97.045,175.056,30.492,155.457
C06126=1073.422,336.421,-97.079,175.059,30.497,155.458
C06127=1073.428,336.669,-97.114,175.063,30.502,155.459
C06128=1073.434,336.916,-97.148,175.066,30.508,155.460
C06129=1073.440,337.164,-97.182,175.069,30.513,155.461
C06130=1073.447,337.412,-97.217,175.073,30.518,155.462
C06131=1073.453,337.659,-97.251,175.076,30.523,155.463
C06132=1073.459,337.907,-97.286,175.080,30.528,155.464
C06133=1073.465,338.154,-97.320,175.082,30.532,155.465
C06134=1073.472,338.401,-97.355,175.086,30.538,155.466
C06135=1073.477,338.649,-97.390,175.089,30.543,155.467
C06136=1073.484,338.897,-97.424,175.093,30.548,155.467
C06137=1073.490,339.144,-97.459,175.096,30.553,155.468
C06138=1073.496,339.391,-97.493,175.099,30.558,155.469
C06139=1073.502,339.640,-97.528,175.103,30.563,155.470
C06140=1073.508,339.886,-97.563,175.106,30.568,155.471
C06141=1073.515,340.134,-97.598,175.110,30.574,155.472
C06142=1073.521,340.382,-97.633,175.112,30.579,155.473
C06143=1073.526,340.629,-97.667,175.116,30.584,155.474
C06144=1073.533,340.877,-97.702,175.120,30.589,155.475
C06145=1073.540,341.125,-97.737,175.123,30.594,155.476
C06146=1073.546,341.371,-97.772,175.127,30.600,155.477
C06147=1073.552,341.620,-97.807,175.129,30.604,155.478
C06148=1073.558,341.867,-97.842,175.133,30.610,155.479
C06149=1073.564,342.114,-97.876,175.136,30.615,155.480
C06150=1073.571,342.362,-97.911,175.140,30.620,155.481
C06151=1073.577,342.609,-97.947,175.144,30.625,155.482
C06152=1073.583,342.857,-97.981,175.147,30.630,155.483
C06153=1073.590,343.104,-98.016,175.150,30.636,155.484
C06154=1073.596,343.352,-98.052,175.153,30.641,155.485
C06155=1073.602,343.600,-98.086,175.157,30.646,155.486
C06156=1073.608,343.846,-98.121,175.160,30.651,155.487
C06157=1073.614,344.063,-98.152,175.163,30.656,155.488
C06158=1073.619,344.279,-98.182,175.167,30.660,155.488
C06159=1073.625,344.496,-98.214,175.169,30.665,155.489
C06160=1073.630,344.711,-98.244,175.172,30.670,155.490
C06161=1073.635,344.929,-98.274,175.176,30.674,155.491
C06162=1073.641,345.144,-98.305,175.178,30.679,155.492
C06163=1073.647,345.361,-98.336,175.182,30.684,155.493
C06164=1073.651,345.577,-98.367,175.184,30.688,155.494
C06165=1073.658,345.825,-98.402,175.188,30.694,155.495
C06166=1073.664,346.072,-98.438,175.192,30.699,155.496
C06167=1073.671,346.320,-98.473,175.195,30.704,155.497
C06168=1073.676,346.567,-98.508,175.198,30.710,155.498
C06169=1073.683,346.814,-98.543,175.201,30.715,155.499
C06170=1073.689,347.062,-98.579,175.205,30.721,155.500
C06171=1073.696,347.309,-98.614,175.208,30.726,155.501
C06172=1073.702,347.557,-98.650,175.212,30.731,155.502
C06173=1073.709,347.804,-98.685,175.216,30.737,155.503
C06174=1073.714,348.051,-98.720,175.219,30.742,155.504
C06175=1073.721,348.298,-98.755,175.223,30.748,155.505
C06176=1073.727,348.546,-98.791,175.226,30.753,155.506
C06177=1073.733,348.794,-98.827,175.230,30.759,155.507
C06178=1073.740,349.041,-98.862,175.232,30.764,155.508
C06179=1073.746,349.289,-98.898,175.236,30.769,155.509
C06180=1073.752,349.536,-98.934,175.240,30.775,155.510
C06181=1073.758,349.783,-98.969,175.243,30.780,155.511
C06182=1073.764,350.030,-99.005,175.247,30.786,155.512
C06183=1073.770,350.278,-99.040,175.250,30.791,155.513
C06184=1073.777,350.525,-99.076,175.254,30.797,155.514
C06185=1073.783,350.772,-99.112,175.258,30.802,155.515
C06186=1073.790,351.020,-99.147,175.261,30.808,155.516
C06187=1073.796,351.267,-99.183,175.265,30.813,155.517
C06188=1073.803,351.514,-99.219,175.268,30.819,155.518
C06189=1073.809,351.762,-99.254,175.272,30.824,155.519
C06190=1073.815,352.009,-99.290,175.275,30.830,155.520
C06191=1073.822,352.257,-99.327,175.279,30.835,155.521
C06192=1073.828,352.504,-99.362,175.283,30.841,155.522
C06193=1073.835,352.752,-99.398,175.286,30.847,155.524
C06194=1073.841,352.999,-99.434,175.290,30.852,155.525
C06195=1073.847,353.246,-99.470,175.293,30.857,155.526
C06196=1073.853,353.493,-99.506,175.297,30.863,155.527
C06197=1073.859,353.741,-99.542,175.301,30.869,155.528
C06198=1073.866,353.988,-99.578,175.304,30.874,155.529
C06199=1073.872,354.236,-99.614,175.308,30.880,155.530
C06200=1073.879,354.483,-99.650,175.310,30.886,155.531
C06201=1073.885,354.730,-99.686,175.314,30.891,155.532
C06202=1073.891,354.977,-99.722,175.318,30.897,155.533
C06203=1073.897,355.224,-99.759,175.321,30.903,155.534
C06204=1073.903,355.472,-99.794,175.325,30.909,155.535
C06205=1073.910,355.719,-99.831,175.328,30.914,155.536
C06206=1073.916,355.966,-99.867,175.333,30.920,155.538
C06207=1073.922,356.214,-99.903,175.336,30.926,155.539
C06208=1073.928,356.461,-99.939,175.340,30.932,155.540
C06209=1073.935,356.708,-99.976,175.344,30.937,155.541
C06210=1073.941,356.956,-100.012,175.347,30.943,155.542
C06211=1073.948,357.203,-100.048,175.351,30.948,155.543
C06212=1073.954,357.450,-100.085,175.354,30.954,155.544
C06213=1073.960,357.668,-100.116,175.357,30.959,155.545
C06214=1073.965,357.886,-100.149,175.361,30.965,155.546
C06215=1073.971,358.104,-100.181,175.363,30.969,155.547
C06216=1073.977,358.322,-100.212,175.367,30.975,155.548
C06217=1073.983,358.541,-100.245,175.371,30.980,155.549
C06218=1073.988,358.759,-100.277,175.373,30.985,155.550
C06219=1073.994,358.976,-100.309,175.377,30.990,155.551
C06220=1073.999,359.195,-100.342,175.380,30.995,155.552
C06221=1074.006,359.442,-100.378,175.383,31.001,155.553
C06222=1074.012,359.689,-100.414,175.387,31.007,155.554
C06223=1074.018,359.936,-100.451,175.390,31.013,155.556
C06224=1074.025,360.183,-100.487,175.395,31.019,155.557
C06225=1074.032,360.431,-100.524,175.399,31.025,155.558
C06226=1074.038,360.678,-100.561,175.402,31.031,155.559
C06227=1074.044,360.925,-100.597,175.406,31.037,155.560
C06228=1074.050,361.172,-100.634,175.409,31.042,155.561
C06229=1074.057,361.419,-100.672,175.413,31.048,155.563
C06230=1074.064,361.666,-100.708,175.417,31.054,155.564
C06231=1074.070,361.914,-100.744,175.420,31.060,155.565
C06232=1074.076,362.161,-100.781,175.424,31.066,155.566
C06233=1074.083,362.408,-100.818,175.427,31.072,155.567
C06234=1074.089,362.656,-100.855,175.431,31.078,155.568
C06235=1074.095,362.902,-100.892,175.436,31.084,155.569
C06236=1074.102,363.149,-100.928,175.439,31.090,155.571
C06237=1074.109,363.397,-100.965,175.443,31.096,155.572
C06238=1074.115,363.644,-101.003,175.446,31.102,155.573
C06239=1074.121,363.891,-101.039,175.450,31.108,155.574
C06240=1074.128,364.139,-101.076,175.454,31.114,155.575
C06241=1074.135,364.385,-101.113,175.457,31.120,155.577
C06242=1074.140,364.632,-101.150,175.461,31.126,155.578
C06243=1074.147,364.880,-101.187,175.465,31.133,155.579
C06244=1074.154,365.127,-101.224,175.469,31.138,155.580
C06245=1074.160,365.375,-101.262,175.473,31.145,155.581
C06246=1074.167,365.621,-101.299,175.476,31.151,155.583
C06247=1074.172,365.868,-101.336,175.480,31.157,155.584
C06248=1074.179,366.116,-101.373,175.483,31.163,155.585
C06249=1074.186,366.362,-101.411,175.487,31.170,155.586
C06250=1074.192,366.609,-101.448,175.492,31.176,155.587
C06251=1074.199,366.856,-101.485,175.495,31.182,155.589
C06252=1074.205,367.104,-101.522,175.499,31.188,155.590
C06253=1074.211,367.350,-101.559,175.503,31.195,155.591
C06254=1074.218,367.598,-101.598,175.506,31.201,155.592
C06255=1074.224,367.845,-101.634,175.511,31.207,155.594
C06256=1074.231,368.092,-101.672,175.514,31.214,155.595
C06257=1074.237,368.339,-101.709,175.518,31.220,155.596
C06258=1074.244,368.586,-101.747,175.522,31.226,155.597
C06259=1074.250,368.833,-101.784,175.525,31.232,155.599
C06260=1074.256,369.080,-101.822,175.530,31.238,155.600
C06261=1074.263,369.327,-101.859,175.533,31.245,155.601
C06262=1074.269,369.574,-101.897,175.537,31.251,155.602
C06263=1074.276,369.821,-101.934,175.541,31.258,155.604
C06264=1074.282,370.068,-101.971,175.544,31.264,155.605
C06265=1074.288,370.316,-102.010,175.549,31.270,155.606
C06266=1074.295,370.562,-102.047,175.553,31.277,155.608
C06267=1074.302,370.810,-102.085,175.556,31.283,155.609
C06268=1074.309,371.057,-102.122,175.560,31.290,155.610
C06269=1074.315,371.324,-102.164,175.564,31.297,155.612
C06270=1074.323,371.592,-102.204,175.569,31.304,155.613
C06271=1074.329,371.859,-102.245,175.573,31.310,155.614
C06272=1074.337,372.126,-102.286,175.577,31.317,155.616
C06273=1074.344,372.373,-102.324,175.581,31.324,155.617
C06274=1074.350,372.620,-102.361,175.585,31.330,155.618
C06275=1074.357,372.867,-102.400,175.589,31.337,155.620
C06276=1074.363,373.114,-102.437,175.593,31.343,155.621
C06277=1074.370,373.361,-102.475,175.596,31.350,155.622
C06278=1074.376,373.608,-102.513,175.600,31.357,155.624
C06279=1074.383,373.855,-102.551,175.605,31.363,155.625
C06280=1074.389,374.102,-102.590,175.608,31.370,155.626
C06281=1074.396,374.348,-102.627,175.612,31.376,155.628
C06282=1074.402,374.596,-102.665,175.616,31.383,155.629
C06283=1074.409,374.843,-102.704,175.620,31.390,155.630
C06284=1074.415,375.089,-102.741,175.624,31.396,155.632
C06285=1074.422,375.337,-102.780,175.628,31.403,155.633
C06286=1074.428,375.584,-102.818,175.632,31.410,155.634
C06287=1074.434,375.831,-102.856,175.636,31.417,155.636
C06288=1074.441,376.077,-102.895,175.639,31.423,155.637
C06289=1074.448,376.324,-102.932,175.644,31.430,155.638
C06290=1074.455,376.571,-102.971,175.648,31.437,155.640
C06291=1074.461,376.818,-103.009,175.651,31.444,155.641
C06292=1074.468,377.065,-103.048,175.656,31.450,155.642
C06293=1074.474,377.312,-103.086,175.660,31.457,155.644
C06294=1074.481,377.558,-103.124,175.663,31.464,155.645
C06295=1074.487,377.806,-103.163,175.668,31.471,155.647
C06296=1074.494,378.053,-103.201,175.672,31.477,155.648
C06297=1074.501,378.300,-103.240,175.675,31.484,155.649
C06298=1074.507,378.546,-103.278,175.680,31.491,155.651
C06299=1074.513,378.793,-103.317,175.684,31.498,155.652
C06300=1074.520,379.040,-103.356,175.687,31.505,155.654
C06301=1074.527,379.287,-103.393,175.692,31.512,155.655
C06302=1074.534,379.534,-103.432,175.696,31.519,155.656
C06303=1074.540,379.780,-103.471,175.700,31.526,155.658
C06304=1074.547,380.027,-103.509,175.704,31.533,155.659
C06305=1074.554,380.274,-103.548,175.708,31.540,155.661
C06306=1074.561,380.521,-103.586,175.712,31.547,155.662
C06307=1074.567,380.768,-103.625,175.716,31.553,155.664
C06308=1074.574,381.015,-103.664,175.721,31.561,155.665
C06309=1074.580,381.231,-103.698,175.724,31.567,155.666
C06310=1074.586,381.446,-103.732,175.727,31.573,155.667
C06311=1074.592,381.662,-103.766,175.731,31.579,155.669
C06312=1074.598,381.879,-103.800,175.734,31.585,155.670
C06313=1074.603,382.094,-103.834,175.738,31.591,155.671
C06314=1074.609,382.311,-103.868,175.742,31.597,155.673
C06315=1074.615,382.527,-103.902,175.746,31.604,155.674
C06316=1074.621,382.743,-103.936,175.749,31.610,155.675
C06317=1074.627,382.989,-103.976,175.753,31.617,155.677
C06318=1074.633,383.236,-104.014,175.758,31.625,155.678
C06319=1074.640,383.483,-104.053,175.761,31.632,155.680
C06320=1074.647,383.730,-104.092,175.765,31.639,155.681
C06321=1074.653,383.977,-104.131,175.770,31.646,155.683
C06322=1074.660,384.224,-104.170,175.773,31.653,155.684
C06323=1074.667,384.470,-104.210,175.778,31.661,155.686
C06324=1074.673,384.717,-104.249,175.782,31.668,155.687
C06325=1074.679,384.958,-104.287,175.786,31.675,155.689
C06326=1074.686,385.199,-104.326,175.790,31.682,155.690
C06327=1074.693,385.439,-104.364,175.794,31.690,155.692
C06328=1074.700,385.681,-104.403,175.798,31.697,155.693
C06329=1074.706,385.922,-104.441,175.802,31.704,155.695
C06330=1074.713,386.162,-104.480,175.807,31.711,155.696
C06331=1074.719,386.403,-104.518,175.811,31.718,155.698
C06332=1074.726,386.645,-104.556,175.814,31.725,155.699
C06333=1074.733,386.891,-104.595,175.819,31.733,155.701
C06334=1074.739,387.138,-104.635,175.823,31.740,155.702
C06335=1074.746,387.384,-104.674,175.827,31.748,155.704
C06336=1074.752,387.631,-104.714,175.832,31.755,155.705
C06337=1074.759,387.878,-104.753,175.836,31.762,155.707
C06338=1074.766,388.124,-104.792,175.840,31.770,155.708
C06339=1074.773,388.372,-104.833,175.844,31.777,155.710
C06340=1074.780,388.618,-104.872,175.849,31.785,155.712
C06341=1074.787,388.865,-104.911,175.853,31.793,155.713
C06342=1074.794,389.111,-104.951,175.857,31.800,155.715
C06343=1074.800,389.358,-104.990,175.861,31.808,155.716
C06344=1074.807,389.605,-105.031,175.866,31.815,155.718
C06345=1074.814,389.851,-105.070,175.870,31.823,155.720
C06346=1074.822,390.098,-105.110,175.874,31.831,155.721
C06347=1074.828,390.344,-105.150,175.879,31.838,155.723
C06348=1074.835,390.592,-105.189,175.883,31.846,155.724
C06349=1074.842,390.838,-105.229,175.887,31.853,155.726
C06350=1074.849,391.084,-105.269,175.892,31.861,155.728
C06351=1074.855,391.331,-105.309,175.896,31.869,155.729
C06352=1074.863,391.578,-105.349,175.901,31.877,155.731
C06353=1074.869,391.824,-105.389,175.905,31.885,155.732
C06354=1074.876,392.071,-105.429,175.909,31.893,155.734
C06355=1074.883,392.317,-105.469,175.914,31.900,155.736
C06356=1074.890,392.564,-105.509,175.917,31.908,155.737
C06357=1074.896,392.811,-105.549,175.922,31.916,155.739
C06358=1074.903,393.057,-105.589,175.927,31.924,155.741
C06359=1074.910,393.304,-105.629,175.931,31.932,155.742
C06360=1074.917,393.551,-105.670,175.935,31.940,155.744
C06361=1074.924,393.797,-105.709,175.940,31.948,155.746
C06362=1074.931,394.044,-105.750,175.944,31.956,155.748
C06363=1074.937,394.290,-105.791,175.949,31.964,155.749
C06364=1074.944,394.537,-105.831,175.953,31.972,155.751
C06365=1074.952,394.783,-105.871,175.957,31.979,155.753
C06366=1074.958,395.030,-105.911,175.962,31.987,155.754
C06367=1074.965,395.276,-105.952,175.967,31.996,155.756
C06368=1074.972,395.523,-105.992,175.970,32.004,155.758
C06369=1074.979,395.770,-106.033,175.975,32.012,155.759
C06370=1074.985,396.016,-106.073,175.980,32.020,155.761
C06371=1074.993,396.263,-106.113,175.985,32.028,155.763
C06372=1074.999,396.509,-106.154,175.988,32.036,155.765
C06373=1075.007,396.756,-106.195,175.993,32.044,155.766
C06374=1075.013,397.003,-106.235,175.998,32.053,155.768
C06375=1075.020,397.249,-106.276,176.002,32.061,155.770
C06376=1075.027,397.496,-106.316,176.006,32.069,155.772
C06377=1075.034,397.742,-106.358,176.011,32.078,155.774
C06378=1075.040,397.989,-106.398,176.016,32.086,155.775
C06379=1075.048,398.235,-106.438,176.020,32.094,155.777
C06380=1075.056,398.482,-106.480,176.025,32.102,155.779
C06381=1075.062,398.732,-106.521,176.029,32.111,155.781
C06382=1075.069,398.983,-106.563,176.034,32.119,155.783
C06383=1075.076,399.232,-106.604,176.039,32.128,155.784
C06384=1075.083,399.483,-106.646,176.044,32.137,155.786
C06385=1075.090,399.730,-106.686,176.047,32.145,155.788
C06386=1075.097,399.976,-106.727,176.052,32.154,155.790
C06387=1075.104,400.223,-106.768,176.057,32.162,155.792
C06388=1075.111,400.469,-106.810,176.062,32.170,155.794
C06389=1075.118,400.715,-106.851,176.067,32.179,155.796
C06390=1075.125,400.962,-106.892,176.070,32.188,155.797
C06391=1075.132,401.209,-106.932,176.075,32.196,155.799
C06392=1075.139,401.456,-106.974,176.080,32.205,155.801
C06393=1075.145,401.702,-107.015,176.085,32.214,155.803
C06394=1075.153,401.948,-107.056,176.090,32.222,155.805
C06395=1075.160,402.195,-107.097,176.095,32.231,155.807
C06396=1075.167,402.442,-107.139,176.098,32.239,155.809
C06397=1075.174,402.688,-107.180,176.103,32.248,155.810
C06398=1075.181,402.934,-107.221,176.108,32.257,155.812
C06399=1075.188,403.180,-107.263,176.113,32.266,155.814
C06400=1075.195,403.427,-107.305,176.118,32.274,155.816
C06401=1075.203,403.674,-107.346,176.122,32.283,155.818
C06402=1075.210,403.920,-107.387,176.127,32.292,155.820
C06403=1075.216,404.166,-107.428,176.132,32.301,155.822
C06404=1075.223,404.412,-107.470,176.137,32.310,155.824
C06405=1075.231,404.659,-107.512,176.142,32.319,155.826
C06406=1075.237,404.906,-107.553,176.147,32.328,155.828
C06407=1075.245,405.152,-107.595,176.150,32.337,155.830
C06408=1075.252,405.398,-107.637,176.155,32.346,155.832
C06409=1075.259,405.645,-107.678,176.160,32.355,155.834
C06410=1075.266,405.891,-107.720,176.165,32.364,155.836
C06411=1075.273,406.138,-107.762,176.170,32.373,155.838
C06412=1075.280,406.384,-107.804,176.175,32.382,155.840
C06413=1075.287,406.630,-107.845,176.180,32.391,155.842
C06414=1075.294,406.876,-107.888,176.184,32.400,155.844
C06415=1075.301,407.123,-107.929,176.189,32.410,155.846
C06416=1075.308,407.369,-107.971,176.194,32.419,155.848
C06417=1075.315,407.616,-108.014,176.199,32.428,155.850
C06418=1075.322,407.862,-108.055,176.204,32.437,155.852
C06419=1075.329,408.108,-108.098,176.209,32.447,155.854
C06420=1075.337,408.354,-108.140,176.214,32.456,155.856
C06421=1075.343,408.601,-108.181,176.219,32.466,155.858
C06422=1075.351,408.847,-108.223,176.224,32.474,155.860
C06423=1075.358,409.094,-108.266,176.228,32.484,155.862
C06424=1075.365,409.341,-108.309,176.234,32.494,155.864
C06425=1075.373,409.587,-108.351,176.239,32.503,155.866
C06426=1075.380,409.833,-108.393,176.244,32.513,155.869
C06427=1075.386,410.080,-108.435,176.249,32.522,155.871
C06428=1075.394,410.326,-108.477,176.254,32.531,155.873
C06429=1075.401,410.572,-108.520,176.259,32.541,155.875
C06430=1075.407,410.818,-108.562,176.264,32.551,155.877
C06431=1075.415,411.064,-108.604,176.269,32.560,155.879
C06432=1075.423,411.311,-108.647,176.274,32.570,155.881
C06433=1075.430,411.557,-108.690,176.280,32.579,155.883
C06434=1075.437,411.803,-108.732,176.284,32.589,155.886
C06435=1075.444,412.049,-108.775,176.289,32.599,155.888
C06436=1075.451,412.295,-108.817,176.294,32.609,155.890
C06437=1075.460,412.549,-108.861,176.299,32.618,155.892
C06438=1075.467,412.803,-108.905,176.305,32.629,155.894
C06439=1075.475,413.056,-108.949,176.310,32.639,155.897
C06440=1075.482,413.310,-108.993,176.316,32.649,155.899
C06441=1075.489,413.556,-109.036,176.321,32.659,155.901
C06442=1075.496,413.802,-109.078,176.326,32.668,155.903
C06443=1075.504,414.048,-109.121,176.331,32.678,155.905
C06444=1075.511,414.295,-109.164,176.337,32.688,155.908
C06445=1075.518,414.541,-109.206,176.342,32.698,155.910
C06446=1075.526,414.787,-109.249,176.347,32.708,155.912
C06447=1075.533,415.033,-109.292,176.352,32.718,155.914
C06448=1075.541,415.280,-109.336,176.358,32.728,155.917
C06449=1075.548,415.525,-109.379,176.363,32.739,155.919
C06450=1075.555,415.772,-109.421,176.368,32.748,155.921
C06451=1075.563,416.018,-109.465,176.374,32.759,155.924
C06452=1075.570,416.264,-109.508,176.379,32.769,155.926
C06453=1075.577,416.511,-109.551,176.384,32.779,155.928
C06454=1075.585,416.756,-109.594,176.389,32.789,155.930
C06455=1075.592,417.003,-109.638,176.395,32.800,155.933
C06456=1075.600,417.248,-109.681,176.400,32.810,155.935
C06457=1075.606,417.495,-109.724,176.406,32.821,155.938
C06458=1075.614,417.741,-109.767,176.411,32.831,155.940
C06459=1075.621,417.987,-109.811,176.416,32.841,155.942
C06460=1075.629,418.233,-109.854,176.422,32.852,155.945
C06461=1075.636,418.479,-109.898,176.427,32.862,155.947
C06462=1075.644,418.725,-109.941,176.433,32.873,155.949
C06463=1075.652,418.971,-109.985,176.438,32.883,155.952
C06464=1075.658,419.217,-110.029,176.443,32.894,155.954
C06465=1075.666,419.464,-110.072,176.449,32.904,155.957
C06466=1075.673,419.709,-110.116,176.454,32.915,155.959
C06467=1075.681,419.955,-110.160,176.460,32.926,155.961
C06468=1075.689,420.201,-110.204,176.466,32.936,155.964
C06469=1075.696,420.447,-110.247,176.472,32.947,155.966
C06470=1075.704,420.693,-110.290,176.477,32.958,155.969
C06471=1075.712,420.940,-110.334,176.483,32.969,155.971
C06472=1075.719,421.185,-110.378,176.488,32.979,155.974
C06473=1075.726,421.432,-110.422,176.494,32.990,155.976
C06474=1075.734,421.678,-110.466,176.499,33.001,155.979
C06475=1075.742,421.924,-110.510,176.505,33.012,155.981
C06476=1075.748,422.170,-110.554,176.510,33.023,155.984
C06477=1075.756,422.415,-110.598,176.516,33.034,155.986
C06478=1075.764,422.662,-110.642,176.522,33.045,155.989
C06479=1075.771,422.907,-110.687,176.528,33.056,155.991
C06480=1075.779,423.153,-110.731,176.534,33.068,155.994
C06481=1075.787,423.399,-110.775,176.539,33.078,155.996
C06482=1075.794,423.645,-110.819,176.545,33.090,155.999
C06483=1075.802,423.891,-110.864,176.550,33.101,156.002
C06484=1075.809,424.137,-110.908,176.556,33.112,156.004
C06485=1075.817,424.383,-110.952,176.563,33.124,156.007
C06486=1075.824,424.629,-110.997,176.568,33.135,156.009
C06487=1075.832,424.875,-111.041,176.574,33.146,156.012
C06488=1075.840,425.120,-111.086,176.580,33.158,156.015
C06489=1075.847,425.367,-111.130,176.585,33.169,156.017
C06490=1075.855,425.613,-111.174,176.591,33.180,156.020
C06491=1075.863,425.859,-111.219,176.598,33.192,156.023
C06492=1075.870,426.104,-111.263,176.603,33.203,156.025
C06493=1075.879,426.375,-111.313,176.610,33.216,156.028
C06494=1075.887,426.646,-111.363,176.616,33.229,156.031
C06495=1075.896,426.918,-111.411,176.623,33.241,156.034
C06496=1075.904,427.189,-111.461,176.630,33.254,156.037
C06497=1075.913,427.435,-111.505,176.636,33.266,156.040
C06498=1075.920,427.681,-111.551,176.641,33.278,156.043
C06499=1075.928,427.926,-111.595,176.648,33.289,156.045
C06500=1075.936,428.172,-111.640,176.654,33.302,156.048
C06501=1075.943,428.418,-111.686,176.660,33.313,156.051
C06502=1075.951,428.664,-111.731,176.666,33.325,156.054
C06503=1075.959,428.910,-111.775,176.672,33.337,156.056
C06504=1075.966,429.155,-111.821,176.678,33.349,156.059
C06505=1075.974,429.401,-111.866,176.684,33.361,156.062
C06506=1075.982,429.646,-111.911,176.691,33.373,156.065
C06507=1075.989,429.892,-111.956,176.697,33.385,156.068
C06508=1075.998,430.138,-112.002,176.703,33.397,156.071
C06509=1076.005,430.384,-112.047,176.710,33.410,156.073
C06510=1076.013,430.630,-112.092,176.716,33.422,156.076
C06511=1076.021,430.875,-112.137,176.721,33.434,156.079
C06512=1076.029,431.120,-112.183,176.728,33.446,156.082
C06513=1076.037,431.367,-112.229,176.734,33.459,156.085
C06514=1076.044,431.613,-112.274,176.740,33.471,156.088
C06515=1076.053,431.858,-112.319,176.747,33.483,156.091
C06516=1076.061,432.104,-112.365,176.753,33.496,156.094
C06517=1076.068,432.349,-112.411,176.759,33.508,156.097
C06518=1076.076,432.595,-112.456,176.766,33.521,156.100
C06519=1076.084,432.840,-112.502,176.772,33.534,156.103
C06520=1076.092,433.086,-112.548,176.779,33.546,156.106
C06521=1076.100,433.332,-112.594,176.785,33.559,156.109
C06522=1076.107,433.577,-112.639,176.791,33.571,156.112
C06523=1076.116,433.823,-112.686,176.798,33.584,156.115
C06524=1076.123,434.068,-112.732,176.804,33.597,156.118
C06525=1076.131,434.314,-112.777,176.811,33.610,156.121
C06526=1076.139,434.560,-112.823,176.818,33.623,156.124
C06527=1076.147,434.805,-112.870,176.825,33.635,156.127
C06528=1076.156,435.051,-112.916,176.831,33.649,156.130
C06529=1076.163,435.296,-112.961,176.838,33.661,156.133
C06530=1076.171,435.542,-113.009,176.844,33.675,156.136
C06531=1076.179,435.787,-113.054,176.851,33.688,156.139
C06532=1076.187,436.033,-113.101,176.857,33.700,156.142
C06533=1076.195,436.278,-113.147,176.864,33.714,156.146
C06534=1076.203,436.524,-113.193,176.871,33.727,156.149
C06535=1076.211,436.769,-113.240,176.878,33.740,156.152
C06536=1076.220,437.015,-113.286,176.884,33.753,156.155
C06537=1076.227,437.260,-113.332,176.891,33.767,156.158
C06538=1076.236,437.505,-113.379,176.898,33.780,156.162
C06539=1076.245,437.751,-113.426,176.905,33.793,156.165
C06540=1076.251,437.996,-113.472,176.912,33.807,156.168
C06541=1076.260,438.242,-113.519,176.918,33.821,156.171
C06542=1076.269,438.487,-113.565,176.926,33.834,156.174
C06543=1076.276,438.732,-113.612,176.932,33.847,156.178
C06544=1076.285,438.978,-113.658,176.939,33.861,156.181
C06545=1076.294,439.223,-113.705,176.947,33.875,156.184
C06546=1076.301,439.469,-113.752,176.953,33.888,156.188
C06547=1076.309,439.714,-113.799,176.960,33.903,156.191
C06548=1076.317,439.959,-113.847,176.968,33.916,156.194
C06549=1076.326,440.223,-113.897,176.974,33.931,156.198
C06550=1076.335,440.488,-113.948,176.982,33.946,156.202
C06551=1076.344,440.752,-113.998,176.990,33.961,156.205
C06552=1076.353,441.017,-114.049,176.998,33.976,156.209
C06553=1076.362,441.261,-114.096,177.005,33.991,156.213
C06554=1076.370,441.507,-114.144,177.012,34.005,156.216
C06555=1076.378,441.752,-114.191,177.020,34.019,156.219
C06556=1076.386,441.998,-114.239,177.026,34.033,156.223
C06557=1076.395,442.243,-114.286,177.034,34.048,156.226
C06558=1076.403,442.489,-114.333,177.041,34.062,156.230
C06559=1076.412,442.734,-114.381,177.049,34.076,156.233
C06560=1076.420,442.979,-114.429,177.056,34.090,156.237
C06561=1076.428,443.224,-114.476,177.063,34.105,156.240
C06562=1076.436,443.469,-114.524,177.070,34.120,156.244
C06563=1076.445,443.714,-114.571,177.078,34.134,156.248
C06564=1076.453,443.960,-114.619,177.085,34.149,156.251
C06565=1076.462,444.204,-114.667,177.093,34.163,156.255
C06566=1076.470,444.450,-114.715,177.101,34.178,156.258
C06567=1076.478,444.695,-114.763,177.108,34.193,156.262
C06568=1076.487,444.940,-114.810,177.115,34.208,156.266
C06569=1076.495,445.185,-114.858,177.123,34.223,156.269
C06570=1076.504,445.430,-114.906,177.130,34.238,156.273
C06571=1076.512,445.675,-114.954,177.138,34.253,156.277
C06572=1076.521,445.921,-115.002,177.146,34.268,156.281
C06573=1076.530,446.166,-115.051,177.153,34.283,156.284
C06574=1076.538,446.411,-115.099,177.161,34.298,156.288
C06575=1076.546,446.656,-115.147,177.169,34.313,156.292
C06576=1076.556,446.901,-115.195,177.176,34.328,156.296
C06577=1076.564,447.146,-115.243,177.183,34.344,156.299
C06578=1076.572,447.391,-115.292,177.190,34.359,156.303
C06579=1076.580,447.636,-115.340,177.197,34.374,156.307
C06580=1076.590,447.881,-115.389,177.203,34.389,156.311
C06581=1076.598,448.126,-115.437,177.209,34.404,156.315
C06582=1076.606,448.371,-115.485,177.215,34.419,156.318
C06583=1076.616,448.615,-115.534,177.221,34.434,156.322
C06584=1076.624,448.859,-115.582,177.226,34.450,156.326
C06585=1076.635,449.104,-115.630,177.231,34.464,156.330
C06586=1076.646,449.349,-115.676,177.236,34.478,156.333
C06587=1076.660,449.595,-115.723,177.241,34.491,156.337
C06588=1076.674,449.841,-115.767,177.246,34.504,156.340
C06589=1076.315,449.837,-116.002,177.225,34.660,156.381
C06590=1076.301,449.590,-115.957,177.221,34.648,156.378
C06591=1076.287,449.345,-115.911,177.216,34.634,156.375
C06592=1076.275,449.100,-115.863,177.210,34.621,156.371
C06593=1076.265,448.856,-115.817,177.204,34.606,156.368
C06594=1076.256,448.610,-115.768,177.199,34.592,156.364
C06595=1076.247,448.366,-115.720,177.193,34.576,156.360
C06596=1076.238,448.121,-115.671,177.188,34.561,156.356
C06597=1076.230,447.877,-115.622,177.181,34.546,156.352
C06598=1076.221,447.632,-115.574,177.174,34.531,156.348
C06599=1076.212,447.387,-115.526,177.167,34.516,156.345
C06600=1076.203,447.142,-115.477,177.161,34.500,156.341
C06601=1076.195,446.897,-115.428,177.153,34.485,156.337
C06602=1076.186,446.652,-115.381,177.146,34.470,156.333
C06603=1076.178,446.407,-115.333,177.138,34.455,156.329
C06604=1076.169,446.162,-115.284,177.130,34.440,156.326
C06605=1076.161,445.917,-115.236,177.123,34.425,156.322
C06606=1076.152,445.671,-115.188,177.115,34.410,156.318
C06607=1076.143,445.427,-115.139,177.107,34.395,156.315
C06608=1076.135,445.181,-115.091,177.100,34.380,156.311
C06609=1076.127,444.936,-115.043,177.092,34.365,156.307
C06610=1076.118,444.691,-114.996,177.084,34.350,156.303
C06611=1076.110,444.446,-114.948,177.077,34.335,156.300
C06612=1076.102,444.201,-114.900,177.069,34.321,156.296
C06613=1076.092,443.955,-114.852,177.061,34.305,156.292
C06614=1076.084,443.710,-114.804,177.054,34.291,156.289
C06615=1076.075,443.465,-114.756,177.046,34.276,156.285
C06616=1076.067,443.220,-114.708,177.039,34.262,156.282
C06617=1076.058,442.975,-114.661,177.031,34.248,156.278
C06618=1076.050,442.730,-114.613,177.024,34.233,156.275
C06619=1076.042,442.484,-114.566,177.016,34.219,156.271
C06620=1076.034,442.239,-114.518,177.009,34.204,156.268
C06621=1076.025,441.994,-114.471,177.002,34.190,156.264
C06622=1076.017,441.749,-114.423,176.995,34.176,156.261
C06623=1076.008,441.504,-114.376,176.987,34.162,156.257
C06624=1076.000,441.258,-114.328,176.980,34.148,156.254
C06625=1075.992,441.014,-114.281,176.972,34.133,156.250
C06626=1075.983,440.766,-114.234,176.965,34.119,156.247
C06627=1075.975,440.519,-114.186,176.958,34.105,156.243
C06628=1075.967,440.273,-114.139,176.951,34.091,156.240
C06629=1075.958,440.025,-114.092,176.943,34.077,156.237
C06630=1075.951,439.780,-114.044,176.936,34.063,156.233
C06631=1075.942,439.535,-113.997,176.930,34.050,156.230
C06632=1075.934,439.289,-113.950,176.922,34.036,156.226
C06633=1075.926,439.044,-113.903,176.915,34.022,156.223
C06634=1075.917,438.799,-113.856,176.908,34.009,156.220
C06635=1075.909,438.553,-113.810,176.901,33.995,156.217
C06636=1075.900,438.308,-113.763,176.894,33.981,156.213
C06637=1075.892,438.063,-113.717,176.887,33.968,156.210
C06638=1075.885,437.817,-113.669,176.881,33.955,156.207
C06639=1075.876,437.571,-113.623,176.873,33.941,156.203
C06640=1075.868,437.327,-113.576,176.866,33.928,156.200
C06641=1075.860,437.081,-113.530,176.860,33.915,156.197
C06642=1075.851,436.835,-113.484,176.853,33.901,156.194
C06643=1075.843,436.590,-113.437,176.846,33.888,156.191
C06644=1075.835,436.345,-113.390,176.839,33.875,156.188
C06645=1075.827,436.099,-113.345,176.832,33.862,156.184
C06646=1075.819,435.853,-113.297,176.826,33.849,156.181
C06647=1075.811,435.607,-113.251,176.819,33.836,156.178
C06648=1075.803,435.362,-113.205,176.813,33.822,156.175
C06649=1075.796,435.117,-113.159,176.805,33.810,156.172
C06650=1075.787,434.872,-113.113,176.798,33.796,156.169
C06651=1075.779,434.626,-113.067,176.792,33.784,156.166
C06652=1075.771,434.381,-113.020,176.785,33.771,156.163
C06653=1075.763,434.135,-112.975,176.779,33.758,156.159
C06654=1075.755,433.889,-112.929,176.772,33.745,156.156
C06655=1075.747,433.644,-112.883,176.766,33.732,156.153
C06656=1075.739,433.399,-112.837,176.759,33.720,156.150
C06657=1075.731,433.153,-112.791,176.753,33.707,156.147
C06658=1075.724,432.907,-112.745,176.746,33.694,156.144
C06659=1075.715,432.661,-112.699,176.740,33.682,156.141
C06660=1075.708,432.416,-112.653,176.733,33.669,156.138
C06661=1075.700,432.170,-112.608,176.727,33.657,156.135
C06662=1075.692,431.925,-112.562,176.720,33.644,156.132
C06663=1075.684,431.679,-112.516,176.714,33.632,156.130
C06664=1075.677,431.433,-112.470,176.707,33.619,156.127
C06665=1075.668,431.188,-112.425,176.701,33.607,156.124
C06666=1075.660,430.942,-112.379,176.695,33.595,156.121
C06667=1075.653,430.696,-112.334,176.688,33.583,156.118
C06668=1075.645,430.450,-112.289,176.682,33.570,156.115
C06669=1075.637,430.205,-112.244,176.675,33.558,156.112
C06670=1075.628,429.959,-112.198,176.669,33.546,156.109
C06671=1075.621,429.713,-112.153,176.664,33.534,156.106
C06672=1075.613,429.468,-112.107,176.657,33.522,156.104
C06673=1075.605,429.222,-112.063,176.651,33.510,156.101
C06674=1075.598,428.977,-112.017,176.645,33.498,156.098
C06675=1075.590,428.730,-111.972,176.638,33.486,156.095
C06676=1075.583,428.485,-111.927,176.632,33.474,156.092
C06677=1075.574,428.239,-111.882,176.626,33.462,156.090
C06678=1075.566,427.993,-111.836,176.620,33.450,156.087
C06679=1075.559,427.747,-111.791,176.614,33.438,156.084
C06680=1075.551,427.501,-111.747,176.607,33.427,156.081
C06681=1075.544,427.255,-111.702,176.601,33.415,156.079
C06682=1075.534,426.983,-111.652,176.595,33.402,156.076
C06683=1075.526,426.711,-111.602,176.588,33.390,156.073
C06684=1075.517,426.437,-111.552,176.581,33.377,156.070
C06685=1075.509,426.164,-111.504,176.575,33.364,156.067
C06686=1075.501,425.919,-111.458,176.569,33.352,156.064
C06687=1075.493,425.673,-111.414,176.563,33.341,156.061
C06688=1075.485,425.427,-111.369,176.557,33.329,156.059
C06689=1075.478,425.181,-111.324,176.551,33.318,156.056
C06690=1075.470,424.936,-111.280,176.546,33.307,156.053
C06691=1075.463,424.689,-111.236,176.539,33.295,156.051
C06692=1075.455,424.443,-111.191,176.533,33.284,156.048
C06693=1075.447,424.197,-111.147,176.528,33.273,156.045
C06694=1075.440,423.952,-111.102,176.522,33.262,156.043
C06695=1075.432,423.706,-111.058,176.515,33.250,156.040
C06696=1075.425,423.460,-111.014,176.510,33.239,156.038
C06697=1075.417,423.214,-110.970,176.504,33.228,156.035
C06698=1075.409,422.968,-110.925,176.499,33.217,156.032
C06699=1075.402,422.722,-110.881,176.492,33.205,156.030
C06700=1075.394,422.476,-110.837,176.486,33.195,156.027
C06701=1075.387,422.230,-110.792,176.481,33.183,156.025
C06702=1075.379,421.984,-110.749,176.475,33.172,156.022
C06703=1075.372,421.739,-110.705,176.470,33.162,156.020
C06704=1075.365,421.492,-110.660,176.464,33.151,156.017
C06705=1075.357,421.246,-110.617,176.458,33.140,156.015
C06706=1075.349,421.000,-110.572,176.452,33.129,156.012
C06707=1075.342,420.755,-110.529,176.447,33.118,156.010
C06708=1075.334,420.508,-110.485,176.441,33.107,156.007
C06709=1075.326,420.262,-110.441,176.436,33.097,156.005
C06710=1075.319,420.017,-110.398,176.430,33.086,156.003
C06711=1075.312,419.770,-110.354,176.424,33.076,156.000
C06712=1075.304,419.524,-110.310,176.418,33.065,155.998
C06713=1075.296,419.279,-110.266,176.413,33.054,155.995
C06714=1075.289,419.032,-110.222,176.408,33.044,155.993
C06715=1075.281,418.786,-110.179,176.402,33.033,155.990
C06716=1075.274,418.540,-110.136,176.397,33.023,155.988
C06717=1075.266,418.294,-110.092,176.391,33.012,155.986
C06718=1075.259,418.048,-110.049,176.386,33.002,155.983
C06719=1075.251,417.802,-110.005,176.381,32.991,155.981
C06720=1075.244,417.556,-109.962,176.374,32.981,155.978
C06721=1075.236,417.310,-109.918,176.369,32.971,155.976
C06722=1075.229,417.064,-109.876,176.363,32.960,155.974
C06723=1075.222,416.817,-109.832,176.358,32.950,155.971
C06724=1075.215,416.571,-109.788,176.353,32.940,155.969
C06725=1075.207,416.325,-109.745,176.347,32.930,155.967
C06726=1075.200,416.079,-109.701,176.342,32.919,155.964
C06727=1075.193,415.832,-109.658,176.337,32.909,155.962
C06728=1075.186,415.587,-109.615,176.332,32.899,155.960
C06729=1075.178,415.341,-109.572,176.326,32.889,155.958
C06730=1075.170,415.094,-109.530,176.321,32.878,155.955
C06731=1075.163,414.849,-109.486,176.316,32.868,155.953
C06732=1075.156,414.602,-109.443,176.310,32.859,155.951
C06733=1075.148,414.356,-109.400,176.305,32.849,155.949
C06734=1075.141,414.109,-109.357,176.300,32.839,155.946
C06735=1075.133,413.864,-109.315,176.295,32.829,155.944
C06736=1075.126,413.617,-109.272,176.289,32.819,155.942
C06737=1075.119,413.370,-109.229,176.284,32.809,155.940
C06738=1075.111,413.116,-109.184,176.279,32.799,155.937
C06739=1075.103,412.861,-109.140,176.273,32.789,155.935
C06740=1075.095,412.606,-109.096,176.268,32.779,155.933
C06741=1075.088,412.351,-109.053,176.263,32.769,155.931
C06742=1075.081,412.105,-109.009,176.258,32.759,155.928
C06743=1075.074,411.859,-108.967,176.252,32.749,155.926
C06744=1075.066,411.612,-108.925,176.247,32.739,155.924
C06745=1075.059,411.366,-108.882,176.242,32.730,155.922
C06746=1075.052,411.119,-108.839,176.237,32.720,155.920
C06747=1075.044,410.873,-108.798,176.232,32.710,155.918
C06748=1075.037,410.627,-108.755,176.227,32.701,155.915
C06749=1075.030,410.380,-108.712,176.222,32.692,155.913
C06750=1075.022,410.134,-108.670,176.216,32.682,155.911
C06751=1075.015,409.888,-108.628,176.211,32.672,155.909
C06752=1075.009,409.642,-108.585,176.206,32.663,155.907
C06753=1075.001,409.396,-108.543,176.201,32.654,155.905
C06754=1074.994,409.149,-108.501,176.196,32.644,155.903
C06755=1074.987,408.903,-108.458,176.191,32.635,155.901
C06756=1074.980,408.657,-108.416,176.186,32.625,155.899
C06757=1074.973,408.411,-108.374,176.181,32.616,155.897
C06758=1074.965,408.164,-108.332,176.176,32.607,155.894
C06759=1074.958,407.917,-108.289,176.171,32.597,155.892
C06760=1074.951,407.671,-108.247,176.166,32.588,155.890
C06761=1074.944,407.425,-108.205,176.161,32.579,155.888
C06762=1074.937,407.178,-108.163,176.156,32.570,155.886
C06763=1074.930,406.932,-108.121,176.151,32.560,155.884
C06764=1074.923,406.685,-108.079,176.146,32.551,155.882
C06765=1074.915,406.439,-108.037,176.142,32.542,155.880
C06766=1074.909,406.193,-107.995,176.137,32.533,155.878
C06767=1074.902,405.947,-107.954,176.132,32.524,155.876
C06768=1074.894,405.701,-107.912,176.127,32.515,155.874
C06769=1074.888,405.454,-107.870,176.122,32.506,155.872
C06770=1074.880,405.208,-107.829,176.117,32.497,155.870
C06771=1074.874,404.961,-107.786,176.112,32.487,155.868
C06772=1074.866,404.715,-107.745,176.107,32.478,155.866
C06773=1074.859,404.469,-107.703,176.102,32.470,155.864
C06774=1074.852,404.222,-107.661,176.098,32.461,155.862
C06775=1074.845,403.975,-107.620,176.094,32.452,155.860
C06776=1074.838,403.729,-107.579,176.089,32.443,155.858
C06777=1074.831,403.483,-107.537,176.084,32.435,155.857
C06778=1074.824,403.236,-107.496,176.079,32.426,155.855
C06779=1074.817,402.990,-107.454,176.074,32.417,155.853
C06780=1074.809,402.743,-107.413,176.069,32.408,155.851
C06781=1074.802,402.497,-107.372,176.064,32.399,155.849
C06782=1074.795,402.250,-107.331,176.060,32.391,155.847
C06783=1074.788,402.004,-107.290,176.056,32.382,155.845
C06784=1074.782,401.757,-107.248,176.051,32.373,155.843
C06785=1074.774,401.511,-107.207,176.046,32.365,155.841
C06786=1074.767,401.264,-107.166,176.041,32.356,155.839
C06787=1074.760,401.018,-107.125,176.036,32.347,155.838
C06788=1074.753,400.772,-107.083,176.032,32.339,155.836
C06789=1074.746,400.525,-107.042,176.027,32.330,155.834
C06790=1074.738,400.278,-107.001,176.023,32.322,155.832
C06791=1074.732,400.033,-106.960,176.018,32.313,155.830
C06792=1074.725,399.786,-106.918,176.013,32.305,155.828
C06793=1074.718,399.538,-106.878,176.009,32.297,155.827
C06794=1074.711,399.288,-106.836,176.004,32.288,155.825
C06795=1074.704,399.036,-106.794,175.999,32.279,155.823
C06796=1074.697,398.784,-106.752,175.994,32.271,155.821
C06797=1074.689,398.532,-106.710,175.990,32.262,155.819
C06798=1074.682,398.285,-106.670,175.985,32.254,155.817
C06799=1074.676,398.039,-106.629,175.981,32.245,155.816
C06800=1074.668,397.792,-106.588,175.976,32.237,155.814
C06801=1074.662,397.546,-106.548,175.971,32.229,155.812
C06802=1074.655,397.299,-106.507,175.967,32.221,155.810
C06803=1074.648,397.052,-106.466,175.963,32.212,155.808
C06804=1074.641,396.806,-106.425,175.958,32.204,155.807
C06805=1074.634,396.559,-106.385,175.953,32.196,155.805
C06806=1074.627,396.313,-106.344,175.949,32.188,155.803
C06807=1074.620,396.066,-106.304,175.944,32.180,155.801
C06808=1074.613,395.820,-106.263,175.940,32.172,155.800
C06809=1074.606,395.573,-106.222,175.935,32.163,155.798
C06810=1074.600,395.326,-106.182,175.931,32.155,155.796
C06811=1074.592,395.080,-106.141,175.926,32.147,155.794
C06812=1074.586,394.833,-106.101,175.921,32.139,155.793
C06813=1074.579,394.587,-106.061,175.918,32.131,155.791
C06814=1074.572,394.340,-106.020,175.913,32.123,155.789
C06815=1074.565,394.094,-105.980,175.908,32.115,155.788
C06816=1074.558,393.847,-105.939,175.904,32.107,155.786
C06817=1074.551,393.601,-105.900,175.899,32.099,155.784
C06818=1074.545,393.354,-105.860,175.896,32.091,155.783
C06819=1074.538,393.107,-105.819,175.891,32.083,155.781
C06820=1074.530,392.861,-105.779,175.886,32.075,155.779
C06821=1074.524,392.615,-105.739,175.882,32.068,155.777
C06822=1074.517,392.367,-105.698,175.878,32.060,155.776
C06823=1074.510,392.121,-105.659,175.873,32.052,155.774
C06824=1074.504,391.875,-105.619,175.869,32.044,155.772
C06825=1074.497,391.628,-105.578,175.864,32.036,155.771
C06826=1074.489,391.381,-105.539,175.860,32.028,155.769
C06827=1074.483,391.135,-105.498,175.856,32.020,155.767
C06828=1074.475,390.888,-105.459,175.851,32.013,155.766
C06829=1074.469,390.641,-105.418,175.847,32.005,155.764
C06830=1074.462,390.395,-105.380,175.842,31.998,155.763
C06831=1074.456,390.148,-105.339,175.838,31.990,155.761
C06832=1074.448,389.901,-105.299,175.834,31.982,155.759
C06833=1074.441,389.655,-105.260,175.829,31.975,155.758
C06834=1074.435,389.408,-105.220,175.825,31.967,155.756
C06835=1074.428,389.162,-105.181,175.821,31.959,155.755
C06836=1074.421,388.914,-105.140,175.817,31.952,155.753
C06837=1074.414,388.668,-105.101,175.812,31.945,155.752
C06838=1074.407,388.421,-105.062,175.807,31.937,155.750
C06839=1074.400,388.175,-105.022,175.804,31.929,155.748
C06840=1074.393,387.929,-104.982,175.799,31.922,155.747
C06841=1074.387,387.682,-104.943,175.795,31.914,155.745
C06842=1074.380,387.435,-104.903,175.790,31.907,155.744
C06843=1074.373,387.188,-104.864,175.787,31.900,155.742
C06844=1074.366,386.941,-104.824,175.782,31.892,155.740
C06845=1074.359,386.694,-104.785,175.778,31.885,155.739
C06846=1074.353,386.453,-104.747,175.773,31.878,155.737
C06847=1074.347,386.211,-104.708,175.770,31.870,155.736
C06848=1074.340,385.970,-104.670,175.766,31.863,155.734
C06849=1074.333,385.728,-104.631,175.761,31.856,155.733
C06850=1074.327,385.487,-104.592,175.757,31.849,155.731
C06851=1074.320,385.245,-104.554,175.753,31.842,155.730
C06852=1074.313,385.004,-104.516,175.749,31.834,155.728
C06853=1074.307,384.762,-104.477,175.745,31.827,155.727
C06854=1074.300,384.515,-104.438,175.741,31.820,155.725
C06855=1074.293,384.269,-104.398,175.737,31.812,155.724
C06856=1074.287,384.022,-104.359,175.732,31.805,155.722
C06857=1074.280,383.775,-104.320,175.728,31.798,155.721
C06858=1074.274,383.528,-104.281,175.724,31.791,155.719
C06859=1074.267,383.281,-104.242,175.720,31.784,155.718
C06860=1074.260,383.035,-104.202,175.715,31.777,155.716
C06861=1074.254,382.788,-104.163,175.711,31.769,155.715
C06862=1074.247,382.541,-104.125,175.708,31.762,155.713
C06863=1074.240,382.294,-104.086,175.703,31.755,155.712
C06864=1074.234,382.047,-104.046,175.699,31.748,155.710
C06865=1074.228,381.801,-104.008,175.695,31.740,155.709
C06866=1074.221,381.554,-103.969,175.691,31.733,155.708
C06867=1074.214,381.307,-103.930,175.687,31.727,155.706
C06868=1074.207,381.060,-103.891,175.682,31.720,155.705
C06869=1074.200,380.814,-103.853,175.679,31.713,155.703
C06870=1074.194,380.567,-103.814,175.674,31.706,155.702
C06871=1074.187,380.319,-103.776,175.670,31.699,155.700
C06872=1074.180,380.073,-103.737,175.667,31.692,155.699
C06873=1074.173,379.826,-103.698,175.662,31.685,155.698
C06874=1074.167,379.579,-103.659,175.658,31.678,155.696
C06875=1074.160,379.332,-103.620,175.654,31.671,155.695
C06876=1074.154,379.085,-103.582,175.650,31.664,155.693
C06877=1074.147,378.839,-103.544,175.646,31.657,155.692
C06878=1074.140,378.592,-103.505,175.641,31.650,155.690
C06879=1074.133,378.345,-103.466,175.638,31.643,155.689
C06880=1074.127,378.097,-103.428,175.634,31.637,155.688
C06881=1074.121,377.851,-103.389,175.629,31.630,155.686
C06882=1074.114,377.604,-103.351,175.626,31.623,155.685
C06883=1074.107,377.357,-103.313,175.622,31.616,155.683
C06884=1074.100,377.111,-103.274,175.617,31.609,155.682
C06885=1074.093,376.863,-103.236,175.614,31.602,155.681
C06886=1074.087,376.617,-103.198,175.610,31.596,155.679
C06887=1074.081,376.369,-103.159,175.605,31.589,155.678
C06888=1074.074,376.123,-103.121,175.602,31.582,155.677
C06889=1074.068,375.876,-103.083,175.598,31.576,155.675
C06890=1074.061,375.629,-103.044,175.593,31.569,155.674
C06891=1074.055,375.382,-103.006,175.590,31.562,155.672
C06892=1074.048,375.136,-102.968,175.586,31.555,155.671
C06893=1074.041,374.888,-102.930,175.582,31.549,155.670
C06894=1074.035,374.641,-102.892,175.577,31.542,155.668
C06895=1074.028,374.395,-102.853,175.574,31.535,155.667
C06896=1074.022,374.147,-102.815,175.570,31.529,155.666
C06897=1074.015,373.900,-102.777,175.565,31.522,155.664
C06898=1074.010,373.653,-102.739,175.562,31.516,155.663
C06899=1074.002,373.407,-102.701,175.558,31.509,155.662
C06900=1073.995,373.159,-102.663,175.554,31.502,155.660
C06901=1073.990,372.912,-102.625,175.550,31.496,155.659
C06902=1073.984,372.685,-102.591,175.547,31.490,155.658
C06903=1073.977,372.459,-102.555,175.543,31.484,155.657
C06904=1073.971,372.232,-102.521,175.540,31.478,155.655
C06905=1073.965,372.004,-102.486,175.536,31.472,155.654
C06906=1073.959,371.777,-102.452,175.532,31.466,155.653
C06907=1073.953,371.550,-102.416,175.529,31.460,155.652
C06908=1073.947,371.323,-102.382,175.525,31.454,155.651
C06909=1073.941,371.096,-102.347,175.521,31.448,155.649
C06910=1073.934,370.849,-102.310,175.518,31.442,155.648
C06911=1073.928,370.602,-102.272,175.514,31.435,155.647
C06912=1073.921,370.355,-102.234,175.510,31.429,155.646
C06913=1073.915,370.108,-102.197,175.506,31.423,155.644
C06914=1073.907,369.861,-102.159,175.502,31.416,155.643
C06915=1073.902,369.614,-102.121,175.498,31.410,155.642
C06916=1073.894,369.367,-102.084,175.495,31.404,155.641
C06917=1073.888,369.120,-102.046,175.490,31.397,155.639
C06918=1073.882,368.872,-102.009,175.486,31.391,155.638
C06919=1073.876,368.626,-101.971,175.483,31.385,155.637
C06920=1073.869,368.378,-101.933,175.479,31.378,155.635
C06921=1073.862,368.132,-101.896,175.475,31.372,155.634
C06922=1073.856,367.884,-101.859,175.472,31.366,155.633
C06923=1073.850,367.638,-101.822,175.467,31.359,155.632
C06924=1073.844,367.391,-101.784,175.463,31.353,155.631
C06925=1073.836,367.144,-101.746,175.460,31.347,155.629
C06926=1073.831,366.896,-101.709,175.456,31.341,155.628
C06927=1073.824,366.649,-101.672,175.452,31.335,155.627
C06928=1073.817,366.402,-101.635,175.449,31.328,155.625
C06929=1073.811,366.155,-101.598,175.444,31.322,155.624
C06930=1073.804,365.908,-101.560,175.440,31.316,155.623
C06931=1073.798,365.661,-101.523,175.437,31.310,155.622
C06932=1073.791,365.414,-101.485,175.433,31.303,155.621
C06933=1073.786,365.166,-101.448,175.429,31.297,155.619
C06934=1073.779,364.920,-101.411,175.426,31.291,155.618
C06935=1073.772,364.672,-101.374,175.422,31.285,155.617
C06936=1073.766,364.425,-101.337,175.419,31.279,155.616
C06937=1073.760,364.178,-101.300,175.414,31.273,155.615
C06938=1073.753,363.931,-101.263,175.410,31.267,155.613
C06939=1073.747,363.684,-101.226,175.407,31.261,155.612
C06940=1073.741,363.437,-101.189,175.403,31.255,155.611
C06941=1073.734,363.189,-101.152,175.399,31.249,155.610
C06942=1073.727,362.943,-101.115,175.396,31.243,155.609
C06943=1073.721,362.696,-101.079,175.392,31.237,155.607
C06944=1073.715,362.448,-101.041,175.388,31.231,155.606
C06945=1073.708,362.200,-101.005,175.385,31.225,155.605
C06946=1073.697,361.823,-100.948,175.378,31.215,155.603
C06947=1073.688,361.445,-100.892,175.373,31.206,155.602
C06948=1073.678,361.067,-100.836,175.367,31.198,155.600
C06949=1073.669,360.689,-100.780,175.362,31.189,155.598
C06950=1073.662,360.441,-100.743,175.358,31.183,155.597
C06951=1073.655,360.194,-100.706,175.355,31.177,155.596
C06952=1073.649,359.947,-100.670,175.350,31.171,155.595
C06953=1073.643,359.700,-100.633,175.346,31.165,155.593
C06954=1073.637,359.453,-100.596,175.343,31.159,155.592
C06955=1073.630,359.205,-100.560,175.339,31.153,155.591
C06956=1073.624,358.958,-100.523,175.336,31.147,155.590
C06957=1073.617,358.711,-100.487,175.332,31.141,155.589
C06958=1073.610,358.404,-100.442,175.327,31.134,155.587
C06959=1073.601,358.098,-100.397,175.323,31.127,155.586
C06960=1073.594,357.792,-100.352,175.318,31.120,155.585
C06961=1073.586,357.484,-100.307,175.314,31.113,155.583
C06962=1073.579,357.237,-100.270,175.310,31.107,155.582
C06963=1073.573,356.990,-100.234,175.307,31.101,155.581
C06964=1073.567,356.743,-100.197,175.303,31.095,155.580
C06965=1073.561,356.496,-100.162,175.299,31.090,155.579
C06966=1073.553,356.248,-100.125,175.296,31.084,155.578
C06967=1073.547,356.001,-100.089,175.292,31.078,155.576
C06968=1073.540,355.754,-100.052,175.288,31.072,155.575
C06969=1073.534,355.506,-100.017,175.285,31.066,155.574
C06970=1073.528,355.259,-99.980,175.281,31.061,155.573
C06971=1073.522,355.012,-99.944,175.278,31.056,155.572
C06972=1073.516,354.765,-99.908,175.274,31.050,155.571
C06973=1073.509,354.518,-99.872,175.270,31.044,155.570
C06974=1073.503,354.270,-99.836,175.267,31.038,155.569
C06975=1073.497,354.023,-99.799,175.263,31.033,155.568
C06976=1073.491,353.776,-99.763,175.259,31.027,155.567
C06977=1073.484,353.528,-99.728,175.256,31.021,155.566
C06978=1073.478,353.281,-99.691,175.252,31.016,155.565
C06979=1073.472,353.034,-99.656,175.249,31.010,155.563
C06980=1073.465,352.787,-99.619,175.245,31.004,155.562
C06981=1073.459,352.539,-99.584,175.242,30.999,155.561
C06982=1073.453,352.291,-99.548,175.239,30.994,155.560
C06983=1073.446,352.045,-99.512,175.235,30.988,155.559
C06984=1073.440,351.797,-99.476,175.232,30.982,155.558
C06985=1073.434,351.550,-99.440,175.228,30.977,155.557
C06986=1073.427,351.302,-99.405,175.224,30.971,155.556
C06987=1073.421,351.055,-99.369,175.221,30.966,155.555
C06988=1073.415,350.808,-99.332,175.217,30.960,155.554
C06989=1073.408,350.560,-99.297,175.213,30.955,155.553
C06990=1073.402,350.313,-99.262,175.210,30.949,155.552
C06991=1073.396,350.065,-99.226,175.206,30.944,155.551
C06992=1073.389,349.818,-99.190,175.203,30.939,155.550
C06993=1073.383,349.571,-99.154,175.199,30.933,155.549
C06994=1073.376,349.323,-99.119,175.195,30.928,155.548
C06995=1073.370,349.076,-99.084,175.193,30.922,155.547
C06996=1073.364,348.829,-99.048,175.189,30.917,155.546
C06997=1073.358,348.581,-99.013,175.186,30.911,155.545
C06998=1073.352,348.334,-98.977,175.182,30.906,155.544
C06999=1073.345,348.086,-98.941,175.178,30.900,155.543
C07000=1073.338,347.839,-98.906,175.175,30.895,155.541
C07001=1073.332,347.591,-98.870,175.171,30.889,155.540
C07002=1073.326,347.344,-98.835,175.168,30.884,155.539
C07003=1073.320,347.097,-98.799,175.164,30.878,155.538
C07004=1073.313,346.850,-98.764,175.161,30.873,155.537
C07005=1073.307,346.602,-98.729,175.158,30.868,155.536
C07006=1073.301,346.355,-98.693,175.154,30.863,155.535
C07007=1073.295,346.107,-98.658,175.151,30.857,155.534
C07008=1073.289,345.860,-98.624,175.147,30.852,155.533
C07009=1073.283,345.612,-98.588,175.143,30.846,155.532
C07010=1073.277,345.395,-98.557,175.141,30.842,155.531
C07011=1073.272,345.179,-98.525,175.137,30.837,155.531
C07012=1073.266,344.961,-98.496,175.134,30.832,155.530
C07013=1073.261,344.745,-98.464,175.132,30.828,155.529
C07014=1073.255,344.528,-98.433,175.128,30.823,155.528
C07015=1073.250,344.311,-98.403,175.125,30.819,155.527
C07016=1073.245,344.094,-98.371,175.123,30.814,155.526
C07017=1073.239,343.877,-98.341,175.119,30.809,155.525
C07018=1073.233,343.629,-98.306,175.116,30.804,155.524
C07019=1073.226,343.382,-98.270,175.113,30.799,155.523
C07020=1073.219,343.134,-98.236,175.109,30.794,155.522
C07021=1073.214,342.887,-98.201,175.106,30.788,155.521
C07022=1073.207,342.639,-98.166,175.102,30.783,155.520
C07023=1073.201,342.391,-98.131,175.099,30.778,155.519
C07024=1073.195,342.144,-98.096,175.095,30.773,155.519
C07025=1073.189,341.897,-98.061,175.092,30.768,155.517
C07026=1073.182,341.649,-98.026,175.089,30.763,155.517
C07027=1073.175,341.402,-97.991,175.085,30.758,155.516
C07028=1073.170,341.154,-97.956,175.082,30.752,155.515
C07029=1073.163,340.907,-97.921,175.078,30.747,155.514
C07030=1073.157,340.659,-97.887,175.075,30.742,155.513
C07031=1073.151,340.412,-97.852,175.072,30.737,155.512
C07032=1073.145,340.164,-97.817,175.068,30.731,155.511
C07033=1073.139,339.917,-97.782,175.065,30.726,155.510
C07034=1073.132,339.669,-97.748,175.062,30.722,155.509
C07035=1073.126,339.422,-97.713,175.058,30.716,155.508
C07036=1073.121,339.174,-97.678,175.055,30.711,155.507
C07037=1073.114,338.926,-97.644,175.051,30.706,155.506
C07038=1073.108,338.679,-97.609,175.048,30.701,155.505
C07039=1073.101,338.431,-97.575,175.045,30.696,155.504
C07040=1073.095,338.184,-97.539,175.041,30.691,155.503
C07041=1073.090,337.937,-97.505,175.038,30.685,155.502
C07042=1073.083,337.689,-97.470,175.034,30.680,155.501
C07043=1073.077,337.441,-97.436,175.032,30.675,155.500
C07044=1073.070,337.194,-97.401,175.028,30.670,155.499
C07045=1073.064,336.946,-97.367,175.024,30.665,155.499
C07046=1073.058,336.699,-97.333,175.021,30.660,155.498
C07047=1073.052,336.451,-97.298,175.018,30.655,155.497
C07048=1073.046,336.203,-97.264,175.015,30.650,155.496
C07049=1073.039,335.956,-97.229,175.011,30.645,155.495
C07050=1073.033,335.709,-97.195,175.008,30.640,155.494
C07051=1073.027,335.461,-97.161,175.005,30.635,155.493
C07052=1073.021,335.213,-97.127,175.001,30.630,155.492
C07053=1073.014,334.965,-97.092,174.998,30.625,155.491
C07054=1073.009,334.718,-97.058,174.995,30.621,155.490
C07055=1073.002,334.470,-97.024,174.991,30.616,155.489
C07056=1072.996,334.223,-96.990,174.988,30.611,155.488
C07057=1072.990,333.975,-96.955,174.985,30.606,155.487
C07058=1072.984,333.728,-96.921,174.982,30.601,155.487
C07059=1072.977,333.480,-96.887,174.978,30.596,155.486
C07060=1072.972,333.232,-96.853,174.975,30.591,155.485
C07061=1072.965,332.984,-96.818,174.972,30.586,155.484
C07062=1072.959,332.737,-96.784,174.968,30.581,155.483
C07063=1072.953,332.490,-96.750,174.965,30.576,155.482
C07064=1072.946,332.242,-96.716,174.962,30.571,155.481
C07065=1072.940,331.995,-96.682,174.959,30.566,155.480
C07066=1072.935,331.774,-96.652,174.956,30.562,155.479
C07067=1072.930,331.556,-96.622,174.952,30.557,155.479
C07068=1072.924,331.336,-96.592,174.950,30.553,155.478
C07069=1072.919,331.117,-96.562,174.947,30.549,155.477
C07070=1072.913,330.897,-96.532,174.944,30.544,155.476
C07071=1072.907,330.677,-96.501,174.941,30.540,155.475
C07072=1072.902,330.458,-96.472,174.938,30.536,155.475
C07073=1072.896,330.238,-96.442,174.936,30.532,155.474
C07074=1072.890,329.991,-96.408,174.932,30.527,155.473
C07075=1072.883,329.743,-96.374,174.929,30.522,155.472
C07076=1072.877,329.496,-96.340,174.926,30.517,155.471
C07077=1072.871,329.247,-96.306,174.922,30.512,155.471
C07078=1072.865,329.000,-96.273,174.920,30.508,155.470
C07079=1072.859,328.753,-96.239,174.916,30.503,155.469
C07080=1072.852,328.505,-96.206,174.912,30.498,155.468
C07081=1072.846,328.257,-96.172,174.910,30.494,155.467
C07082=1072.840,328.009,-96.138,174.906,30.489,155.466
C07083=1072.833,327.762,-96.105,174.903,30.484,155.465
C07084=1072.828,327.514,-96.071,174.900,30.479,155.465
C07085=1072.820,327.266,-96.037,174.897,30.474,155.464
C07086=1072.815,327.018,-96.004,174.894,30.470,155.463
C07087=1072.808,326.771,-95.971,174.890,30.465,155.462
C07088=1072.802,326.523,-95.937,174.887,30.461,155.461
C07089=1072.796,326.275,-95.903,174.884,30.456,155.460
C07090=1072.790,326.028,-95.870,174.881,30.451,155.459
C07091=1072.784,325.780,-95.836,174.877,30.446,155.459
C07092=1072.777,325.532,-95.803,174.874,30.441,155.458
C07093=1072.771,325.285,-95.769,174.871,30.437,155.457
C07094=1072.765,325.037,-95.736,174.868,30.432,155.456
C07095=1072.759,324.789,-95.703,174.865,30.428,155.455
C07096=1072.752,324.542,-95.669,174.861,30.422,155.454
C07097=1072.747,324.294,-95.636,174.859,30.418,155.453
C07098=1072.740,324.046,-95.603,174.855,30.413,155.453
C07099=1072.735,323.799,-95.569,174.852,30.409,155.452
C07100=1072.728,323.551,-95.536,174.849,30.404,155.451
C07101=1072.722,323.303,-95.502,174.846,30.399,155.450
C07102=1072.716,323.055,-95.470,174.843,30.394,155.449
C07103=1072.710,322.808,-95.436,174.839,30.390,155.448
C07104=1072.704,322.560,-95.403,174.836,30.386,155.448
C07105=1072.698,322.312,-95.370,174.833,30.381,155.447
C07106=1072.692,322.065,-95.337,174.830,30.376,155.446
C07107=1072.685,321.816,-95.304,174.827,30.371,155.445
C07108=1072.679,321.569,-95.270,174.824,30.367,155.444
C07109=1072.673,321.322,-95.237,174.821,30.362,155.443
C07110=1072.667,321.074,-95.204,174.817,30.357,155.443
C07111=1072.661,320.826,-95.171,174.814,30.353,155.442
C07112=1072.655,320.578,-95.137,174.811,30.348,155.441
C07113=1072.649,320.331,-95.105,174.808,30.344,155.440
C07114=1072.644,320.083,-95.071,174.805,30.339,155.439
C07115=1072.637,319.835,-95.039,174.802,30.334,155.438
C07116=1072.631,319.588,-95.006,174.799,30.330,155.438
C07117=1072.625,319.340,-94.973,174.796,30.325,155.437
C07118=1072.619,319.092,-94.940,174.792,30.320,155.436
C07119=1072.614,318.844,-94.906,174.790,30.315,155.435
C07120=1072.607,318.597,-94.874,174.786,30.311,155.434
C07121=1072.601,318.349,-94.841,174.784,30.307,155.433
C07122=1072.595,318.126,-94.811,174.780,30.302,155.433
C07123=1072.590,317.903,-94.782,174.778,30.298,155.432
C07124=1072.585,317.680,-94.752,174.775,30.294,155.431
C07125=1072.579,317.458,-94.722,174.772,30.290,155.430
C07126=1072.574,317.236,-94.692,174.770,30.286,155.430
C07127=1072.568,317.013,-94.663,174.767,30.281,155.429
C07128=1072.564,316.790,-94.633,174.764,30.278,155.428
C07129=1072.558,316.567,-94.604,174.761,30.273,155.428
C07130=1072.552,316.319,-94.572,174.758,30.269,155.427
C07131=1072.546,316.071,-94.539,174.755,30.264,155.426
C07132=1072.541,315.824,-94.506,174.752,30.259,155.425
C07133=1072.534,315.577,-94.473,174.750,30.255,155.424
C07134=1072.528,315.329,-94.440,174.746,30.251,155.424
C07135=1072.523,315.080,-94.408,174.744,30.246,155.423
C07136=1072.517,314.833,-94.375,174.740,30.241,155.422
C07137=1072.510,314.585,-94.342,174.737,30.237,155.421
C07138=1072.505,314.337,-94.310,174.734,30.232,155.420
C07139=1072.498,314.089,-94.278,174.731,30.228,155.419
C07140=1072.492,313.842,-94.245,174.728,30.223,155.419
C07141=1072.486,313.594,-94.213,174.725,30.219,155.418
C07142=1072.479,313.346,-94.180,174.722,30.214,155.417
C07143=1072.473,313.098,-94.148,174.719,30.210,155.416
C07144=1072.467,312.850,-94.115,174.715,30.206,155.416
C07145=1072.461,312.603,-94.082,174.713,30.201,155.415
C07146=1072.455,312.354,-94.050,174.709,30.197,155.414
C07147=1072.449,312.107,-94.018,174.707,30.192,155.413
C07148=1072.442,311.859,-93.986,174.703,30.188,155.412
C07149=1072.436,311.612,-93.954,174.701,30.183,155.412
C07150=1072.430,311.364,-93.922,174.697,30.179,155.411
C07151=1072.424,311.116,-93.890,174.694,30.175,155.410
C07152=1072.418,310.868,-93.857,174.691,30.171,155.409
C07153=1072.412,310.620,-93.825,174.688,30.166,155.409
C07154=1072.406,310.372,-93.792,174.686,30.162,155.408
C07155=1072.399,310.124,-93.761,174.682,30.157,155.407
C07156=1072.393,309.876,-93.729,174.680,30.153,155.406
C07157=1072.387,309.629,-93.697,174.676,30.148,155.406
C07158=1072.381,309.381,-93.664,174.673,30.144,155.405
C07159=1072.375,309.133,-93.632,174.670,30.140,155.404
C07160=1072.368,308.885,-93.600,174.667,30.136,155.403
C07161=1072.362,308.637,-93.568,174.664,30.131,155.403
C07162=1072.357,308.390,-93.537,174.661,30.127,155.402
C07163=1072.351,308.142,-93.504,174.659,30.122,155.401
C07164=1072.345,307.894,-93.472,174.655,30.118,155.400
C07165=1072.338,307.646,-93.440,174.652,30.113,155.399
C07166=1072.332,307.398,-93.408,174.649,30.109,155.399
C07167=1072.326,307.151,-93.376,174.646,30.105,155.398
C07168=1072.320,306.903,-93.344,174.643,30.100,155.397
C07169=1072.313,306.655,-93.313,174.640,30.096,155.396
C07170=1072.308,306.407,-93.281,174.638,30.092,155.396
C07171=1072.302,306.159,-93.249,174.634,30.087,155.395
C07172=1072.296,305.911,-93.217,174.632,30.083,155.394
C07173=1072.290,305.664,-93.185,174.628,30.079,155.393
C07174=1072.284,305.416,-93.153,174.625,30.074,155.393
C07175=1072.278,305.168,-93.121,174.623,30.070,155.392
C07176=1072.272,304.920,-93.089,174.619,30.065,155.391
C07177=1072.266,304.672,-93.058,174.617,30.061,155.390
C07178=1072.260,304.451,-93.030,174.614,30.057,155.390
C07179=1072.255,304.230,-93.001,174.612,30.053,155.389
C07180=1072.249,304.009,-92.973,174.609,30.050,155.388
C07181=1072.244,303.788,-92.944,174.606,30.046,155.388
C07182=1072.239,303.567,-92.916,174.604,30.042,155.387
C07183=1072.234,303.346,-92.888,174.601,30.038,155.386
C07184=1072.229,303.125,-92.860,174.599,30.034,155.386
C07185=1072.223,302.904,-92.831,174.596,30.030,155.385
C07186=1072.217,302.657,-92.800,174.592,30.026,155.384
C07187=1072.211,302.408,-92.769,174.590,30.022,155.383
C07188=1072.205,302.160,-92.736,174.587,30.018,155.383
C07189=1072.199,301.913,-92.705,174.584,30.013,155.382
C07190=1072.193,301.665,-92.673,174.581,30.009,155.381
C07191=1072.188,301.417,-92.642,174.579,30.004,155.381
C07192=1072.181,301.169,-92.610,174.575,30.000,155.380
C07193=1072.176,300.922,-92.579,174.572,29.996,155.379
C07194=1072.170,300.673,-92.547,174.570,29.992,155.378
C07195=1072.164,300.426,-92.516,174.566,29.987,155.378
C07196=1072.158,300.178,-92.484,174.564,29.983,155.377
C07197=1072.153,299.930,-92.453,174.561,29.979,155.376
C07198=1072.146,299.682,-92.421,174.558,29.974,155.375
C07199=1072.141,299.434,-92.390,174.555,29.970,155.375
C07200=1072.135,299.186,-92.358,174.553,29.965,155.374
C07201=1072.129,298.939,-92.327,174.549,29.961,155.373
C07202=1072.123,298.690,-92.296,174.547,29.957,155.372
C07203=1072.118,298.442,-92.264,174.544,29.953,155.372
C07204=1072.111,298.194,-92.233,174.541,29.948,155.371
C07205=1072.106,297.946,-92.202,174.538,29.944,155.370
C07206=1072.099,297.698,-92.170,174.535,29.940,155.369
C07207=1072.094,297.451,-92.139,174.532,29.935,155.369
C07208=1072.087,297.202,-92.108,174.529,29.931,155.368
C07209=1072.082,296.955,-92.076,174.527,29.927,155.367
C07210=1072.076,296.706,-92.046,174.523,29.922,155.366
C07211=1072.069,296.459,-92.015,174.521,29.919,155.366
C07212=1072.064,296.210,-91.983,174.518,29.914,155.365
C07213=1072.058,295.963,-91.952,174.515,29.910,155.364
C07214=1072.052,295.715,-91.922,174.512,29.906,155.364
C07215=1072.046,295.467,-91.890,174.509,29.902,155.363
C07216=1072.040,295.219,-91.859,174.507,29.897,155.362
C07217=1072.033,294.971,-91.828,174.503,29.893,155.361
C07218=1072.028,294.723,-91.797,174.501,29.889,155.361
C07219=1072.022,294.475,-91.766,174.498,29.885,155.360
C07220=1072.016,294.227,-91.735,174.495,29.881,155.359
C07221=1072.009,293.979,-91.705,174.492,29.877,155.359
C07222=1072.004,293.731,-91.673,174.490,29.872,155.358
C07223=1071.997,293.483,-91.642,174.487,29.868,155.357
C07224=1071.992,293.235,-91.612,174.484,29.864,155.356
C07225=1071.986,292.988,-91.581,174.481,29.860,155.356
C07226=1071.980,292.739,-91.549,174.478,29.856,155.355
C07227=1071.974,292.491,-91.519,174.475,29.851,155.354
C07228=1071.968,292.243,-91.489,174.472,29.847,155.353
C07229=1071.961,291.995,-91.457,174.470,29.843,155.353
C07230=1071.956,291.748,-91.427,174.467,29.839,155.352
C07231=1071.950,291.499,-91.396,174.464,29.835,155.351
C07232=1071.944,291.251,-91.365,174.461,29.830,155.351
C07233=1071.938,291.004,-91.334,174.459,29.826,155.350
C07234=1071.933,290.790,-91.308,174.456,29.823,155.349
C07235=1071.928,290.576,-91.282,174.453,29.819,155.349
C07236=1071.922,290.362,-91.255,174.451,29.815,155.348
C07237=1071.917,290.148,-91.229,174.449,29.812,155.348
C07238=1071.913,289.936,-91.202,174.447,29.808,155.347
C07239=1071.907,289.722,-91.176,174.444,29.805,155.346
C07240=1071.901,289.508,-91.150,174.441,29.801,155.346
C07241=1071.897,289.294,-91.123,174.439,29.797,155.345
C07242=1071.891,289.046,-91.093,174.436,29.794,155.344
C07243=1071.885,288.799,-91.062,174.434,29.790,155.344
C07244=1071.879,288.550,-91.032,174.431,29.785,155.343
C07245=1071.873,288.302,-91.001,174.429,29.781,155.342
C07246=1071.867,288.054,-90.971,174.425,29.777,155.342
C07247=1071.861,287.806,-90.940,174.423,29.773,155.341
C07248=1071.855,287.558,-90.910,174.420,29.769,155.340
C07249=1071.849,287.310,-90.879,174.417,29.765,155.340
C07250=1071.843,287.062,-90.849,174.414,29.761,155.339
C07251=1071.837,286.814,-90.818,174.411,29.757,155.338
C07252=1071.831,286.566,-90.788,174.409,29.753,155.337
C07253=1071.824,286.318,-90.758,174.406,29.748,155.337
C07254=1071.818,286.069,-90.728,174.404,29.744,155.336
C07255=1071.813,285.822,-90.698,174.400,29.740,155.335
C07256=1071.807,285.574,-90.668,174.398,29.736,155.335
C07257=1071.800,285.325,-90.637,174.395,29.732,155.334
